			(* If we lose Side A Clamp PS In the AutoCycle between AC_Clamp and AC_Unclamp we Fault *)
			IF nActiveFaults[2].31=0 AND (nAutoCycleStep > AC_Clamp) AND ( nAutoCycleStep < AC_Unclamp) AND
				NOT bPS617
			THEN
				nActiveFaults[2].31:=1;
				IF (nFaultArrayIndex<=5) THEN
					arrFaultMessage[nFaultArrayIndex]:='F256 - Clamp Pressure Lost - Side A';
					arrFaultWarningCurrent[nCurrent]:='F256 - Clamp Pressure Lost - Side A';
					nFaultArrayIndex:=nFaultArrayIndex+1;
					nCurrent:=nCurrent+1;
				END_IF
			END_IF

		END_IF (*	Side A Faults *)

	(* 	SIDE B FAULTS
		The text of the fault comes from the function block "Side_B_Fixture" and we assign the hundreds series # to it below.
		Example: Side A Fixture has F2 is concated to the front of the text so that they are 200 series faults
				Side B fixture has F3 concated to make them 300 series faults..  
		You must go to the function block to see the rest of the number and the description text of the fault. 
		Generally this will be at the bottom of the function block. 	*)
		IF bSideBEnabled THEN
			(* Tailstock Side A *)
			IF nActiveFaults[3].0=0 AND Side_B_Fixture.bError THEN
				nActiveFaults[3].0:=1;
				IF (nFaultArrayIndex<=5) THEN
					arrFaultMessage[nFaultArrayIndex]:=CONCAT('F3',Side_B_Fixture.sErrorText);
						arrFaultMessage[nFaultArrayIndex]:=CONCAT(arrFaultMessage[nFaultArrayIndex],' Side B');
					arrFaultWarningCurrent[nCurrent]:=CONCAT('F3',Side_B_Fixture.sErrorText);
						arrFaultWarningCurrent[nCurrent]:=CONCAT(arrFaultWarningCurrent[nCurrent],' Side B');
					nCurrent:=nCurrent+1;
					nFaultArrayIndex:=nFaultArrayIndex+1;
					nCurrent:=nCurrent+1;
				END_IF
			END_IF

			IF nActiveFaults[3].1=0 AND bBCoolantSolenoid
				AND bLowFlow1B AND NOT(fCoolantFlowMin<0.5)
				AND fbFlowAverageTimer1BLOW.Q AND fbCoolantOnDelayTON.Q
			THEN
				nActiveFaults[3].1:=1;
				IF (nFaultArrayIndex<=5) THEN
					arrFaultMessage[nFaultArrayIndex]:='F330 - Coolant Flow Below Min #1B';
					arrFaultWarningCurrent[nCurrent]:='F330 - Coolant Flow Below Min #1B';
					nFaultArrayIndex:=nFaultArrayIndex+1;
					nCurrent:=nCurrent+1;
				END_IF
			END_IF
			IF nActiveFaults[3].2=0 AND bBCoolantSolenoid
				AND bHighFlow1B AND NOT(fCoolantFlowMax=60)
				AND fbFlowAverageTimer1BHIGH.Q AND fbCoolantOnDelayTON.Q
			THEN
				nActiveFaults[3].2:=1;
				IF (nFaultArrayIndex<=5) THEN
					arrFaultMessage[nFaultArrayIndex]:='F331 - Coolant Flow Exceeded Max #1B';
					arrFaultWarningCurrent[nCurrent]:='F331 - Coolant Flow Exceeded Max #1B';
					nFaultArrayIndex:=nFaultArrayIndex+1;
					nCurrent:=nCurrent+1;
				END_IF
			END_IF

			IF nActiveFaults[3].3=0 AND bBCoolantSolenoid
				AND bLowFlow2B AND NOT(fCoolantFlowMin<0.5)
				AND fbFlowAverageTimer2BLOW.Q AND fbCoolantOnDelayTON.Q
			THEN
				nActiveFaults[3].3:=1;
				IF (nFaultArrayIndex<=5) THEN
					arrFaultMessage[nFaultArrayIndex]:='F332 - Coolant Flow Below Min #2B';
					arrFaultWarningCurrent[nCurrent]:='F332 - Coolant Flow Below Min #2B';
					nFaultArrayIndex:=nFaultArrayIndex+1;
					nCurrent:=nCurrent+1;
				END_IF
			END_IF
			IF nActiveFaults[3].4=0 AND bBCoolantSolenoid
				AND bHighFlow2B AND NOT(fCoolantFlowMax=60)
				AND fbFlowAverageTimer2BHIGH.Q AND fbCoolantOnDelayTON.Q
			THEN
				nActiveFaults[3].4:=1;
				IF (nFaultArrayIndex<=5) THEN
					arrFaultMessage[nFaultArrayIndex]:='F333 - Coolant Flow Exceeded Max #2B';
					arrFaultWarningCurrent[nCurrent]:='F333 - Coolant Flow Exceeded Max #2B';
					nFaultArrayIndex:=nFaultArrayIndex+1;
					nCurrent:=nCurrent+1;
				END_IF
			END_IF

			IF nActiveFaults[3].5=0 AND bBCoolantSolenoid
				AND bLowFlow3B AND NOT(fCoolantFlowMin<0.5)
				AND fbFlowAverageTimer3BLOW.Q AND fbCoolantOnDelayTON.Q
			THEN
				nActiveFaults[3].5:=1;
				IF (nFaultArrayIndex<=5) THEN
					arrFaultMessage[nFaultArrayIndex]:='F334 - Coolant Flow Below Min #3B';
					arrFaultWarningCurrent[nCurrent]:='F334 - Coolant Flow Below Min #3B';
					nFaultArrayIndex:=nFaultArrayIndex+1;
					nCurrent:=nCurrent+1;
				END_IF
			END_IF
			IF nActiveFaults[3].6=0 AND bBCoolantSolenoid
				AND bHighFlow3B AND NOT(fCoolantFlowMax=60)
				AND fbFlowAverageTimer3BHIGH.Q AND fbCoolantOnDelayTON.Q
			THEN
				nActiveFaults[3].6:=1;
				IF (nFaultArrayIndex<=5) THEN
					arrFaultMessage[nFaultArrayIndex]:='F335 - Coolant Flow Exceeded Max #3B';
					arrFaultWarningCurrent[nCurrent]:='F335 - Coolant Flow Exceeded Max #3B';
					nFaultArrayIndex:=nFaultArrayIndex+1;
					nCurrent:=nCurrent+1;
				END_IF
			END_IF

			IF nActiveFaults[3].7=0 AND NOT(nServoThrustMax=0) AND fbServoBThrustMaxDelayTON.Q
				AND bInCycle AND NOT(stZBAxis.Status.InPositionArea) AND (stZBAxis.NcToPlc.AxisState=3) THEN
				nActiveFaults[3].7:=1;
				IF (nFaultArrayIndex<=5) THEN
					arrFaultMessage[nFaultArrayIndex]:='F336 - Servo ZB Thrust Exceeded Max';
					arrFaultWarningCurrent[nCurrent]:='F336 - Servo  ZBThrust Exceeded Max';
					nFaultArrayIndex:=nFaultArrayIndex+1;
					nCurrent:=nCurrent+1;
				END_IF
			END_IF

			IF nActiveFaults[3].8=0 AND stZBAxis.Status.Error  THEN
				nActiveFaults[3].8:=1;
				IF (nFaultArrayIndex<=5) THEN
					IF nZBAxisDiagNumber=64720 THEN
						arrFaultMessage[nFaultArrayIndex]:='F337a - ZB Negative Overtravel - (-) Motion Disabled';
						arrFaultWarningCurrent[nCurrent]:='F337a - ZB Negative Overtravel - (-) Motion Disabled';
					ELSIF nZBAxisDiagNumber=64721 THEN
						arrFaultMessage[nFaultArrayIndex]:='F337b - ZB Positive Overtravel - (+) Motion Disabled';
						arrFaultWarningCurrent[nCurrent]:='F337b - ZB Positive Overtravel - (+) Motion Disabled';
					ELSE
						arrFaultMessage[nFaultArrayIndex]:=CONCAT('F337 - Servo ZB Axis Fault# ',
							UDINT_TO_STRING(stZBAxis.Status.ErrorID));
						arrFaultWarningCurrent[nCurrent]:=CONCAT('F337 - Servo ZB Axis Fault# ',
							UDINT_TO_STRING(stZBAxis.Status.ErrorID));
					END_IF
					nFaultArrayIndex:=nFaultArrayIndex+1;
					nCurrent:=nCurrent+1;
				END_IF
			END_IF

			IF nActiveFaults[3].9=0 AND stWBAxis.Status.Error  THEN
				nActiveFaults[3].9:=1;
				IF (nFaultArrayIndex<=5) THEN
					IF nWBAxisDiagNumber=64720 THEN
						arrFaultMessage[nFaultArrayIndex]:='F338a - WB Negative Overtravel - (-) Motion Disabled';
						arrFaultWarningCurrent[nCurrent]:='F338a - WB Negative Overtravel - (-) Motion Disabled';
					ELSIF nWBAxisDiagNumber=64721 THEN
						arrFaultMessage[nFaultArrayIndex]:='F338b - WB Positive Overtravel - (+) Motion Disabled';
						arrFaultWarningCurrent[nCurrent]:='F338b - WB Positive Overtravel - (+) Motion Disabled';
					ELSE
						arrFaultMessage[nFaultArrayIndex]:=CONCAT('F338 - Servo WB Axis Fault# ',
							UDINT_TO_STRING(stWBAxis.Status.ErrorID));
						arrFaultWarningCurrent[nCurrent]:=CONCAT('F338 - Servo WB Axis Fault# ',
							UDINT_TO_STRING(stWBAxis.Status.ErrorID));
					END_IF
					nFaultArrayIndex:=nFaultArrayIndex+1;
					nCurrent:=nCurrent+1;
				END_IF
			END_IF

			IF nActiveFaults[3].10=0 AND fbHomeWB.Error  THEN
				nActiveFaults[3].10:=1;
				IF (nFaultArrayIndex<=5) THEN
					arrFaultMessage[nFaultArrayIndex]:='F339 - Tailstock WB Homing Error';
					arrFaultWarningCurrent[nCurrent]:='F339 - Tailstock WB Homing Error';;
					nFaultArrayIndex:=nFaultArrayIndex+1;
					nCurrent:=nCurrent+1;
				END_IF
			END_IF

			IF nActiveFaults[3].11=0 AND nSpindleLoad1BDisplay>nSpindleLoadMax AND NOT(nSpindleLoadMax=0)
				AND bVFD_BRun AND bVFD_B1UpToSpeed AND fbBLoadFaultDelay.Q THEN
				 nActiveFaults[3].11:=1;
				IF (nFaultArrayIndex<=5) THEN
					arrFaultMessage[nFaultArrayIndex]:='F340 - Spindle #1B Max Load Exceeded';
					arrFaultWarningCurrent[nCurrent]:='F340 - Spindle #1B Max Load Exceeded';
					nFaultArrayIndex:=nFaultArrayIndex+1;
					nCurrent:=nCurrent+1;
				END_IF
			END_IF

			IF nActiveFaults[3].12=0 AND nSpindleLoad2BDisplay>nSpindleLoadMax AND NOT(nSpindleLoadMax=0)
				AND bVFD_BRun AND bVFD_B2UpToSpeed AND fbBLoadFaultDelay.Q THEN
				 nActiveFaults[3].12:=1;
				IF (nFaultArrayIndex<=5) THEN
					arrFaultMessage[nFaultArrayIndex]:='F341 - Spindle #2B Max Load Exceeded';
					arrFaultWarningCurrent[nCurrent]:='F341 - Spindle #2B Max Load Exceeded';
					nFaultArrayIndex:=nFaultArrayIndex+1;
					nCurrent:=nCurrent+1;
				END_IF
			END_IF

			IF nActiveFaults[3].13=0 AND nSpindleLoad3BDisplay>nSpindleLoadMax AND NOT(nSpindleLoadMax=0)
				AND bVFD_BRun AND bVFD_B3UpToSpeed AND fbBLoadFaultDelay.Q THEN
				 nActiveFaults[3].13:=1;
				IF (nFaultArrayIndex<=5) THEN
					arrFaultMessage[nFaultArrayIndex]:='F342 - Spindle #3B Max Load Exceeded';
					arrFaultWarningCurrent[nCurrent]:='F342 - Spindle #3B Max Load Exceeded';
					nFaultArrayIndex:=nFaultArrayIndex+1;
					nCurrent:=nCurrent+1;
				END_IF
			END_IF

	(* Spares *)

			IF nActiveFaults[3].18=0 AND fbVFD_B1.bError THEN
			(*	Encompasses ALL VFD related Errors *)
			(* uptospeed, drivenotready, drivefaulted, drivewarning, drivecomm *)
				nActiveFaults[3].18:=1;
				IF (nFaultArrayIndex<=5) THEN
					IF fbVFD_B1.nErrorID=Er_DriveComm THEN
						arrFaultMessage[nFaultArrayIndex]:='F343a - Spindle #1B VFD Communcation Failed';
						arrFaultWarningCurrent[nCurrent]:='F343a - Spindle #1B VFD Communcation Failed';
						nFaultArrayIndex:=nFaultArrayIndex+1;
						nCurrent:=nCurrent+1;
					ELSIF fbVFD_B1.nErrorID=Er_DriveFaulted THEN
						arrFaultMessage[nFaultArrayIndex]:='F343b - Spindle #1B VFD Fault';
						arrFaultWarningCurrent[nCurrent]:='F343b - Spindle #1B VFD Fault';
						nFaultArrayIndex:=nFaultArrayIndex+1;
						nCurrent:=nCurrent+1;
					ELSIF fbVFD_B1.nErrorID=Er_DriveWarning THEN
						arrFaultMessage[nFaultArrayIndex]:='F343c - Spindle #1B VFD Warning';
						arrFaultWarningCurrent[nCurrent]:='F343c - Spindle #1B VFD Warning';
						nFaultArrayIndex:=nFaultArrayIndex+1;
						nCurrent:=nCurrent+1;
					ELSIF fbVFD_B1.nErrorID=Er_DriveNotReady THEN
						arrFaultMessage[nFaultArrayIndex]:='F343d - Spindle #1B VFD Not Ready';
						arrFaultWarningCurrent[nCurrent]:='F343d - Spindle #1B VFD Not Ready';
						nFaultArrayIndex:=nFaultArrayIndex+1;
						nCurrent:=nCurrent+1;
					ELSIF fbVFD_B1.nErrorID=Er_InvalidRPM THEN
						arrFaultMessage[nFaultArrayIndex]:='F343e - Spindle #1B VFD Invalid RPM Requested';
						arrFaultWarningCurrent[nCurrent]:='F343e - Spindle #1B VFD Invalid RPM Requested';
						nFaultArrayIndex:=nFaultArrayIndex+1;
						nCurrent:=nCurrent+1;
					ELSIF fbVFD_B1.nErrorID=Er_InvalidRatio THEN
						arrFaultMessage[nFaultArrayIndex]:='F343f - Spindle #1B VFD Invalid Motor to Spindle Ratio Requested';
						arrFaultWarningCurrent[nCurrent]:='F343f - Spindle #1B VFD Invalid Motor to Spindle Ratio Requested';
						nFaultArrayIndex:=nFaultArrayIndex+1;
						nCurrent:=nCurrent+1;
					ELSIF fbVFD_B1.nErrorID=Er_InvalidOverride THEN
						arrFaultMessage[nFaultArrayIndex]:='F343g - Spindle #1B VFD Invalid Override Requested';
						arrFaultWarningCurrent[nCurrent]:='F343g - Spindle #1B VFD Invalid Override Requested';
						nFaultArrayIndex:=nFaultArrayIndex+1;
						nCurrent:=nCurrent+1;
					ELSIF fbVFD_B1.nErrorID=Er_UpToSpeedTimeout THEN
						arrFaultMessage[nFaultArrayIndex]:='F343h - Spindle #1B VFD Not Up To Speed';
						arrFaultWarningCurrent[nCurrent]:='F343h - Spindle #1B VFD Not Up To Speed';
						nFaultArrayIndex:=nFaultArrayIndex+1;
						nCurrent:=nCurrent+1;
					ELSE
						arrFaultMessage[nFaultArrayIndex]:=CONCAT('F343 - Spindle #1B VFD Error : ',
												UDINT_TO_STRING(fbVFD_B1.stVFDInfo.nActiveFault));
						arrFaultWarningCurrent[nCurrent]:=CONCAT('F343 - Spindle #1B VFD Error : ',
												UDINT_TO_STRING(fbVFD_B1.stVFDInfo.nActiveFault));
						nFaultArrayIndex:=nFaultArrayIndex+1;
						nCurrent:=nCurrent+1;
					END_IF
				END_IF
			END_IF

			IF nActiveFaults[3].19=0 AND fbVFD_B2.bError THEN
			(*	Encompasses ALL VFD related Errors *)
			(* uptospeed, drivenotready, drivefaulted, drivewarning, drivecomm *)
				nActiveFaults[3].19:=1;
				IF (nFaultArrayIndex<=5) THEN
					IF fbVFD_B2.nErrorID=Er_DriveComm THEN
						arrFaultMessage[nFaultArrayIndex]:='F344a - Spindle #2B VFD Communcation Failed';
						arrFaultWarningCurrent[nCurrent]:='F344a - Spindle #2B VFD Communcation Failed';
						nFaultArrayIndex:=nFaultArrayIndex+1;
						nCurrent:=nCurrent+1;
					ELSIF fbVFD_B2.nErrorID=Er_DriveFaulted THEN
						arrFaultMessage[nFaultArrayIndex]:='F344b - Spindle #2B VFD Fault';
						arrFaultWarningCurrent[nCurrent]:='F344b - Spindle #2B VFD Fault';
						nFaultArrayIndex:=nFaultArrayIndex+1;
						nCurrent:=nCurrent+1;
					ELSIF fbVFD_B2.nErrorID=Er_DriveWarning THEN
						arrFaultMessage[nFaultArrayIndex]:='F344c - Spindle #2B VFD Warning';
						arrFaultWarningCurrent[nCurrent]:='F344c - Spindle #2B VFD Warning';
						nFaultArrayIndex:=nFaultArrayIndex+1;
						nCurrent:=nCurrent+1;
					ELSIF fbVFD_B2.nErrorID=Er_DriveNotReady THEN
						arrFaultMessage[nFaultArrayIndex]:='F344d - Spindle #2B VFD Not Ready';
						arrFaultWarningCurrent[nCurrent]:='F344d - Spindle #2B VFD Not Ready';
						nFaultArrayIndex:=nFaultArrayIndex+1;
						nCurrent:=nCurrent+1;
					ELSIF fbVFD_B2.nErrorID=Er_InvalidRPM THEN
						arrFaultMessage[nFaultArrayIndex]:='F344e - Spindle #2B VFD Invalid RPM Requested';
						arrFaultWarningCurrent[nCurrent]:='F344e - Spindle #2B VFD Invalid RPM Requested';
						nFaultArrayIndex:=nFaultArrayIndex+1;
						nCurrent:=nCurrent+1;
					ELSIF fbVFD_B2.nErrorID=Er_InvalidRatio THEN
						arrFaultMessage[nFaultArrayIndex]:='F344f - Spindle #2B VFD Invalid Motor to Spindle Ratio Requested';
						arrFaultWarningCurrent[nCurrent]:='F344f - Spindle #2B VFD Invalid Motor to Spindle Ratio Requested';
						nFaultArrayIndex:=nFaultArrayIndex+1;
						nCurrent:=nCurrent+1;
					ELSIF fbVFD_B2.nErrorID=Er_InvalidOverride THEN
						arrFaultMessage[nFaultArrayIndex]:='F344g - Spindle #2B VFD Invalid Override Requested';
						arrFaultWarningCurrent[nCurrent]:='F344g - Spindle #2B VFD Invalid Override Requested';
						nFaultArrayIndex:=nFaultArrayIndex+1;
						nCurrent:=nCurrent+1;
					ELSIF fbVFD_B2.nErrorID=Er_UpToSpeedTimeout THEN
						arrFaultMessage[nFaultArrayIndex]:='F344h - Spindle #2B VFD Not Up To Speed';
						arrFaultWarningCurrent[nCurrent]:='F344h - Spindle #2B VFD Not Up To Speed';
						nFaultArrayIndex:=nFaultArrayIndex+1;
						nCurrent:=nCurrent+1;
					ELSE
						arrFaultMessage[nFaultArrayIndex]:=CONCAT('F344 - Spindle #2B VFD Error : ',
												UDINT_TO_STRING(fbVFD_B2.stVFDInfo.nActiveFault));
						arrFaultWarningCurrent[nCurrent]:=CONCAT('F344 - Spindle #2B VFD Error : ',
												UDINT_TO_STRING(fbVFD_B2.stVFDInfo.nActiveFault));
						nFaultArrayIndex:=nFaultArrayIndex+1;
						nCurrent:=nCurrent+1;
					END_IF
				END_IF
			END_IF

			IF nActiveFaults[3].20=0 AND fbVFD_B3.bError THEN
			(*	Encompasses ALL VFD related Errors *)
			(* uptospeed, drivenotready, drivefaulted, drivewarning, drivecomm *)
				nActiveFaults[3].20:=1;
				IF (nFaultArrayIndex<=5) THEN
					IF fbVFD_B3.nErrorID=Er_DriveComm THEN
						arrFaultMessage[nFaultArrayIndex]:='F345a - Spindle #3B VFD Communcation Failed';
						arrFaultWarningCurrent[nCurrent]:='F345a - Spindle #3B VFD Communcation Failed';
						nFaultArrayIndex:=nFaultArrayIndex+1;
						nCurrent:=nCurrent+1;
					ELSIF fbVFD_B3.nErrorID=Er_DriveFaulted THEN
						arrFaultMessage[nFaultArrayIndex]:='F345b - Spindle #3B VFD Fault';
						arrFaultWarningCurrent[nCurrent]:='F345b - Spindle #3B VFD Fault';
						nFaultArrayIndex:=nFaultArrayIndex+1;
						nCurrent:=nCurrent+1;
					ELSIF fbVFD_B3.nErrorID=Er_DriveWarning THEN
						arrFaultMessage[nFaultArrayIndex]:='F345c - Spindle #3B VFD Warning';
						arrFaultWarningCurrent[nCurrent]:='F345c - Spindle #3B VFD Warning';
						nFaultArrayIndex:=nFaultArrayIndex+1;
						nCurrent:=nCurrent+1;
					ELSIF fbVFD_B3.nErrorID=Er_DriveNotReady THEN
						arrFaultMessage[nFaultArrayIndex]:='F345d - Spindle #3B VFD Not Ready';
						arrFaultWarningCurrent[nCurrent]:='F345d - Spindle #3B VFD Not Ready';
						nFaultArrayIndex:=nFaultArrayIndex+1;
						nCurrent:=nCurrent+1;
					ELSIF fbVFD_B3.nErrorID=Er_InvalidRPM THEN
						arrFaultMessage[nFaultArrayIndex]:='F345e - Spindle #3B VFD Invalid RPM Requested';
						arrFaultWarningCurrent[nCurrent]:='F345e - Spindle #3B VFD Invalid RPM Requested';
						nFaultArrayIndex:=nFaultArrayIndex+1;
						nCurrent:=nCurrent+1;
					ELSIF fbVFD_B3.nErrorID=Er_InvalidRatio THEN
						arrFaultMessage[nFaultArrayIndex]:='F345f - Spindle #3B VFD Invalid Motor to Spindle Ratio Requested';
						arrFaultWarningCurrent[nCurrent]:='F345f - Spindle #3B VFD Invalid Motor to Spindle Ratio Requested';
						nFaultArrayIndex:=nFaultArrayIndex+1;
						nCurrent:=nCurrent+1;
					ELSIF fbVFD_B3.nErrorID=Er_InvalidOverride THEN
						arrFaultMessage[nFaultArrayIndex]:='F345g - Spindle #3B VFD Invalid Override Requested';
						arrFaultWarningCurrent[nCurrent]:='F345g - Spindle #3B VFD Invalid Override Requested';
						nFaultArrayIndex:=nFaultArrayIndex+1;
						nCurrent:=nCurrent+1;
					ELSIF fbVFD_B3.nErrorID=Er_UpToSpeedTimeout THEN
						arrFaultMessage[nFaultArrayIndex]:='F345h - Spindle #3B VFD Not Up To Speed';
						arrFaultWarningCurrent[nCurrent]:='F345h - Spindle #3B VFD Not Up To Speed';
						nFaultArrayIndex:=nFaultArrayIndex+1;
						nCurrent:=nCurrent+1;
					ELSE
						arrFaultMessage[nFaultArrayIndex]:=CONCAT('F345 - Spindle #3B VFD Error : ',
												UDINT_TO_STRING(fbVFD_B3.stVFDInfo.nActiveFault));
						arrFaultWarningCurrent[nCurrent]:=CONCAT('F345 - Spindle #3B VFD Error : ',
												UDINT_TO_STRING(fbVFD_B3.stVFDInfo.nActiveFault));
						nFaultArrayIndex:=nFaultArrayIndex+1;
						nCurrent:=nCurrent+1;
					END_IF
				END_IF
			END_IF

			(* Coolant Pressure Fault for Auto Mode *)
			IF nActiveFaults[3].21=0 AND fbLowPressureFaultBDelay.Q
				AND bMachineMode
			THEN
				nActiveFaults[3].21:=1;
				IF (nFaultArrayIndex<=5) THEN
					arrFaultMessage[nFaultArrayIndex]:='F346 - Coolant Pressure Low - Side B';
					arrFaultWarningCurrent[nCurrent]:='F346 - Coolant Pressure Low - Side B';
					nFaultArrayIndex:=nFaultArrayIndex+1;
					nCurrent:=nCurrent+1;
				END_IF
			END_IF

			IF nActiveFaults[3].22=0 AND fbSpeedVariationTimer1BHIGH.Q
				AND bVFD_BRun  AND bVFD_B1UpToSpeed AND (bInCycle OR bSetupB)
				AND fbBSpeedDelayTimer.Q THEN
				nActiveFaults[3].22:=1;
				IF (nFaultArrayIndex<=5) THEN
					arrFaultMessage[nFaultArrayIndex]:='F347 - Spindle Speed Not Correct #1B (HIGH)';
					arrFaultWarningCurrent[nCurrent]:='F333 - Spindle Speed Not Correct #1B (HIGH)';
					nFaultArrayIndex:=nFaultArrayIndex+1;
					nCurrent:=nCurrent+1;
				END_IF
			END_IF
			IF nActiveFaults[3].23=0 AND fbSpeedVariationTimer1BLOW.Q
				AND bVFD_BRun AND bVFD_B1UpToSpeed AND (bInCycle OR bSetupB)
				AND fbBSpeedDelayTimer.Q THEN
				nActiveFaults[3].23:=1;
				IF (nFaultArrayIndex<=5) THEN
					arrFaultMessage[nFaultArrayIndex]:='F348 - Spindle Speed Not Correct #1B (LOW)';
					arrFaultWarningCurrent[nCurrent]:='F348 - Spindle Speed Not Correct #1B (LOW)';
					nFaultArrayIndex:=nFaultArrayIndex+1;
					nCurrent:=nCurrent+1;
				END_IF
			END_IF

			IF nActiveFaults[3].24=0 AND fbSpeedVariationTimer2BHIGH.Q
				AND bVFD_BRun  AND bVFD_B2UpToSpeed AND (bInCycle OR bSetupB)
				AND fbBSpeedDelayTimer.Q THEN
				nActiveFaults[3].24:=1;
				IF (nFaultArrayIndex<=5) THEN
					arrFaultMessage[nFaultArrayIndex]:='F349 - Spindle Speed Not Correct #2B (HIGH)';
					arrFaultWarningCurrent[nCurrent]:='F349 - Spindle Speed Not Correct #2B (HIGH)';
					nFaultArrayIndex:=nFaultArrayIndex+1;
					nCurrent:=nCurrent+1;
				END_IF
			END_IF

			IF nActiveFaults[3].25=0 AND fbSpeedVariationTimer2BLOW.Q
				AND bVFD_BRun AND bVFD_B2UpToSpeed AND (bInCycle OR bSetupB)
				AND fbBSpeedDelayTimer.Q THEN
				nActiveFaults[3].25:=1;
				IF (nFaultArrayIndex<=5) THEN
					arrFaultMessage[nFaultArrayIndex]:='F350 - Spindle Speed Not Correct #2B (LOW)';
					arrFaultWarningCurrent[nCurrent]:='F350 - Spindle Speed Not Correct #2B (LOW)';
					nFaultArrayIndex:=nFaultArrayIndex+1;
					nCurrent:=nCurrent+1;
				END_IF
			END_IF

			IF nActiveFaults[3].26=0 AND fbSpeedVariationTimer3BHIGH.Q
				AND bVFD_BRun  AND bVFD_B3UpToSpeed AND (bInCycle OR bSetupB)
				AND fbBSpeedDelayTimer.Q THEN
				nActiveFaults[3].26:=1;
				IF (nFaultArrayIndex<=5) THEN
					arrFaultMessage[nFaultArrayIndex]:='F351 - Spindle Speed Not Correct #3B (HIGH)';
					arrFaultWarningCurrent[nCurrent]:='F351 - Spindle Speed Not Correct #3B (HIGH)';
					nFaultArrayIndex:=nFaultArrayIndex+1;
					nCurrent:=nCurrent+1;
				END_IF
			END_IF

			IF nActiveFaults[3].27=0 AND fbSpeedVariationTimer3BLOW.Q
				AND bVFD_BRun AND bVFD_B3UpToSpeed AND (bInCycle OR bSetupB)
				AND fbBSpeedDelayTimer.Q THEN
				nActiveFaults[3].27:=1;
				IF (nFaultArrayIndex<=5) THEN
					arrFaultMessage[nFaultArrayIndex]:='F352 - Spindle Speed Not Correct #3B (LOW)';
					arrFaultWarningCurrent[nCurrent]:='F352 - Spindle Speed Not Correct #3B (LOW)';
					nFaultArrayIndex:=nFaultArrayIndex+1;
					nCurrent:=nCurrent+1;
				END_IF
			END_IF

			IF nActiveFaults[3].28=0 AND nModeError=Er_SideBColletSolError THEN
				nModeError:=Er_NoModeError;
				nActiveFaults[3].28:=1;
				IF (nFaultArrayIndex<=5) THEN
					arrFaultMessage[nFaultArrayIndex]:='F353 - Both B Clamp and UnClamp Solenoids On At Same Time';
					arrFaultWarningCurrent[nCurrent]:='F353 - Both B Clamp and UnClamp Solenoids On At Same Time';
					nFaultArrayIndex:=nFaultArrayIndex+1;
					nCurrent:=nCurrent+1;
				END_IF
			END_IF

			IF nActiveFaults[3].29=0 AND nModeError=Er_SideBEjectorsSolError THEN
				nModeError:=Er_NoModeError;
				nActiveFaults[3].29:=1;
				IF (nFaultArrayIndex<=5) THEN
					arrFaultMessage[nFaultArrayIndex]:='F354 - Both B Ejector Advance  and Retract Solenoids On At Same Time';
					arrFaultWarningCurrent[nCurrent]:='F354 - Both B Ejector Advance  and Retract Solenoids On At Same Time';
					nFaultArrayIndex:=nFaultArrayIndex+1;
					nCurrent:=nCurrent+1;
				END_IF
			END_IF

			IF nActiveFaults[3].30=0 AND bRack7Comm THEN
				nActiveFaults[3].30:=1;
				IF (nFaultArrayIndex<=5) THEN
					arrFaultMessage[nFaultArrayIndex]:='F355 - Com. Lost to Side B Tailstock Input Module';
					arrFaultWarningCurrent[nCurrent]:='F355 - Com. Lost to Side B Tailstock Input Module';
					nFaultArrayIndex:=nFaultArrayIndex+1;
					nCurrent:=nCurrent+1;
				END_IF
			END_IF

			(* If we lose Side B Clamp PS In the AutoCycle between AC_Clamp and AC_Unclamp we Fault *)
			IF nActiveFaults[3].31=0 AND (nAutoCycleStep > AC_Clamp) AND (nAutoCycleStep < AC_Unclamp) AND
				NOT bPS727
			THEN
				nActiveFaults[3].31:=1;
				IF (nFaultArrayIndex<=5) THEN
					arrFaultMessage[nFaultArrayIndex]:='F356 - Clamp Pressure Lost - Side B';
					arrFaultWarningCurrent[nCurrent]:='F356 - Clamp Pressure Lost - Side B';
					nFaultArrayIndex:=nFaultArrayIndex+1;
					nCurrent:=nCurrent+1;
				END_IF
			END_IF

		END_IF (*	Side B Faults *)

	(* Faults that do not Stop a Drilling Cycle *)

		IF nActiveFaults[4].0=0 AND bFilter1Dirty AND nDirtyCount1=5 THEN
			nActiveFaults[4].0:=1;
			IF (nFaultArrayIndex<=5) THEN
				arrFaultMessage[nFaultArrayIndex]:='F400 - Filter #1 Clogged (MUST CHANGE)';
				arrFaultWarningCurrent[nCurrent]:='F400 - Filter #1 Clogged (MUST CHANGE)';
				nFaultArrayIndex:=nFaultArrayIndex+1;
				nCurrent:=nCurrent+1;
			END_IF
		END_IF

		IF nActiveFaults[4].1=0 AND bFilter2Dirty AND nDirtyCount2=5 THEN
			nActiveFaults[4].1:=1;
			IF (nFaultArrayIndex<=5) THEN
				arrFaultMessage[nFaultArrayIndex]:='F401 - Filter #2 Clogged (MUST CHANGE)';
				arrFaultWarningCurrent[nCurrent]:='F401 - Filter #2 Clogged (MUST CHANGE)';
				nFaultArrayIndex:=nFaultArrayIndex+1;
				nCurrent:=nCurrent+1;
			END_IF
		END_IF

		IF nActiveFaults[4].2=0 AND bFilter3Dirty AND nDirtyCount3=5 THEN
			nActiveFaults[4].2:=1;
			IF (nFaultArrayIndex<=5) THEN
				arrFaultMessage[nFaultArrayIndex]:='F402 - Filter #3 Clogged (MUST CHANGE)';
				arrFaultWarningCurrent[nCurrent]:='F402 - Filter #3 Clogged (MUST CHANGE)';
				nFaultArrayIndex:=nFaultArrayIndex+1;
				nCurrent:=nCurrent+1;
			END_IF
		END_IF

		IF nActiveFaults[4].3=0 AND bFilter4Dirty AND nDirtyCount4=5 THEN
			nActiveFaults[4].3:=1;
			IF (nFaultArrayIndex<=5) THEN
				arrFaultMessage[nFaultArrayIndex]:='F403 - Filter #4 Clogged (MUST CHANGE)';
				arrFaultWarningCurrent[nCurrent]:='F403 - Filter #4 Clogged (MUST CHANGE)';
				nFaultArrayIndex:=nFaultArrayIndex+1;
				nCurrent:=nCurrent+1;
			END_IF
		END_IF

		IF nActiveFaults[4].4=0 AND NOT(bLubeLevel) AND (nLubeLevelLowCount>=3) THEN
			nActiveFaults[4].4:=1;
			IF (nFaultArrayIndex<=5) THEN
				arrFaultMessage[nFaultArrayIndex]:='F404 - Lube Level Low (MUST FILL)';
				arrFaultWarningCurrent[nCurrent]:='F404 - Lube Level Low (MUST FILL)';
				nFaultArrayIndex:=nFaultArrayIndex+1;
				nCurrent:=nCurrent+1;
			END_IF
		END_IF

		(* Fault if Side A Collet Clamped and X selected on MPG *)
		IF nActiveFaults[4].5=0 AND ( ( (bPS617 OR bATailstockColletClamp) AND bXAAxisSelected) OR
			( (bPS727 OR bBTailstockColletClamp) AND bXBAxisSelected) ) THEN
			nActiveFaults[4].5:=1;
			IF (nFaultArrayIndex<=5) THEN
				IF bXAAxisSelected THEN
					arrFaultMessage[nFaultArrayIndex]:='F405A - MPG XA Selected While Clamped';
					arrFaultWarningCurrent[nCurrent]:='F405A - MPG XA Selected While Clamped';
				ELSE
					arrFaultMessage[nFaultArrayIndex]:='F405B - MPG XB Selected While Clamped';
					arrFaultWarningCurrent[nCurrent]:='F405B - MPG XB Selected While Clamped';
				END_IF
				nFaultArrayIndex:=nFaultArrayIndex+1;
				nCurrent:=nCurrent+1;
			END_IF
		END_IF

		(* Fault if Side A Collet Clamped and ZA or WA selected on MPG *)
		IF nActiveFaults[4].6=0 AND (bPS617 OR bATailstockColletClamp) AND (bZAAxisSelected OR bWAAxisSelected) THEN
			nActiveFaults[4].6:=1;
			IF (nFaultArrayIndex<=5) THEN
				arrFaultMessage[nFaultArrayIndex]:='F406 - MPG ZA or WA Selected While Clamped';
				arrFaultWarningCurrent[nCurrent]:='F406 - MPG ZA or WA Selected While Clamped';
				nFaultArrayIndex:=nFaultArrayIndex+1;
				nCurrent:=nCurrent+1;
			END_IF
		END_IF

		(* Fault if Side B Collet Clamped and ZB or WB selected on MPG *)
		IF nActiveFaults[4].7=0 AND (bPS727 OR bBTailstockColletClamp) AND (bZBAxisSelected OR bWBAxisSelected) THEN
			nActiveFaults[4].7:=1;
			IF (nFaultArrayIndex<=5) THEN
				arrFaultMessage[nFaultArrayIndex]:='F407 - MPG ZB or WB Selected While Clamped';
				arrFaultWarningCurrent[nCurrent]:='F407 - MPG ZB or WB Selected While Clamped';
				nFaultArrayIndex:=nFaultArrayIndex+1;
				nCurrent:=nCurrent+1;
			END_IF
		END_IF

	(* 	WARNINGS		*)

		IF nActiveWarnings[1].0=0 AND fbCoolantTempWarningTON.Q THEN
			nActiveWarnings[1].0:=1;
			IF (nWarningArrayIndex<=5) THEN
				arrFaultMessage[nWarningArrayIndex+5]:='W001 - Coolant Temperature Warning';
				arrFaultWarningCurrent[nCurrent]:='W001 - Coolant Temperature Warning';
				nWarningArrayIndex:=nWarningArrayIndex+1;
				nCurrent:=nCurrent+1;
			END_IF
		ELSIF NOT( bCoolantTempWarning) AND nActiveWarnings[1].0=1 THEN
			IF FIND(arrFaultMessage[6], 'W001')>0 THEN
				arrFaultMessage[6]:=arrFaultMessage[7];
				arrFaultMessage[7]:=arrFaultMessage[8];
				arrFaultMessage[8]:=arrFaultMessage[9];
				arrFaultMessage[9]:=arrFaultMessage[10];
				arrFaultMessage[10]:='';
				nActiveWarnings[1].0:=0;
				nWarningArrayIndex:=nWarningArrayIndex-1;
			ELSIF FIND(arrFaultMessage[7], 'W001')>0 THEN
				arrFaultMessage[7]:=arrFaultMessage[8];
				arrFaultMessage[8]:=arrFaultMessage[9];
				arrFaultMessage[9]:=arrFaultMessage[10];
				arrFaultMessage[10]:='';
				nActiveWarnings[1].0:=0;
				nWarningArrayIndex:=nWarningArrayIndex-1;
			ELSIF FIND(arrFaultMessage[8], 'W001')>0 THEN
				arrFaultMessage[8]:=arrFaultMessage[9];
				arrFaultMessage[9]:=arrFaultMessage[10];
				arrFaultMessage[10]:='';
				nActiveWarnings[1].0:=0;
				nWarningArrayIndex:=nWarningArrayIndex-1;
			ELSIF FIND(arrFaultMessage[9], 'W001')>0 THEN
				arrFaultMessage[9]:=arrFaultMessage[10];
				arrFaultMessage[10]:='';
				nActiveWarnings[1].0:=0;
				nWarningArrayIndex:=nWarningArrayIndex-1;
			ELSIF FIND(arrFaultMessage[10], 'W001')>0 THEN
				arrFaultMessage[10]:='';
				nActiveWarnings[1].0:=0;
				nWarningArrayIndex:=nWarningArrayIndex-1;
			ELSE
				nActiveWarnings[1].0:=0;
				nWarningArrayIndex:=nWarningArrayIndex-1;
			END_IF
		END_IF

		IF nActiveWarnings[1].1=0 AND NOT(bProx310)
			AND (bMachineMode OR bEnterAutoModePB) AND NOT(bInCycle) THEN
			nActiveWarnings[1].1:=1;
			IF (nWarningArrayIndex<=5) THEN
				arrFaultMessage[nWarningArrayIndex+5]:='W002 - Tool Change Door Open Side A';
				arrFaultWarningCurrent[nCurrent]:='W002 - Tool Change Door Open Side A';
				nWarningArrayIndex:=nWarningArrayIndex+1;
				nCurrent:=nCurrent+1;
			END_IF
		ELSIF bProx310 AND nActiveWarnings[1].1 THEN
			IF FIND(arrFaultMessage[6], 'W002')>0 THEN
				arrFaultMessage[6]:=arrFaultMessage[7];
				arrFaultMessage[7]:=arrFaultMessage[8];
				arrFaultMessage[8]:=arrFaultMessage[9];
				arrFaultMessage[9]:=arrFaultMessage[10];
				arrFaultMessage[10]:='';
				nActiveWarnings[1].1:=0;
				nWarningArrayIndex:=nWarningArrayIndex-1;
			ELSIF FIND(arrFaultMessage[7], 'W002')>0 THEN
				arrFaultMessage[7]:=arrFaultMessage[8];
				arrFaultMessage[8]:=arrFaultMessage[9];
				arrFaultMessage[9]:=arrFaultMessage[10];
				arrFaultMessage[10]:='';
				nActiveWarnings[1].1:=0;
				nWarningArrayIndex:=nWarningArrayIndex-1;
			ELSIF FIND(arrFaultMessage[8], 'W002')>0 THEN
				arrFaultMessage[8]:=arrFaultMessage[9];
				arrFaultMessage[9]:=arrFaultMessage[10];
				arrFaultMessage[10]:='';
				nActiveWarnings[1].1:=0;
				nWarningArrayIndex:=nWarningArrayIndex-1;
			ELSIF FIND(arrFaultMessage[9], 'W002')>0 THEN
				arrFaultMessage[9]:=arrFaultMessage[10];
				arrFaultMessage[10]:='';
				nActiveWarnings[1].1:=0;
				nWarningArrayIndex:=nWarningArrayIndex-1;
			ELSIF FIND(arrFaultMessage[10], 'W002')>0 THEN
				arrFaultMessage[10]:='';
				nActiveWarnings[1].1:=0;
				nWarningArrayIndex:=nWarningArrayIndex-1;
			ELSE
				nActiveWarnings[1].1:=0;
				nWarningArrayIndex:=nWarningArrayIndex-1;
			END_IF
		END_IF

		IF nActiveWarnings[1].2=0 AND NOT(bProx312)
			AND (bMachineMode OR bEnterAutoModePB) AND NOT(bInCycle) THEN
			nActiveWarnings[1].2:=1;
			IF (nWarningArrayIndex<=5) THEN
				arrFaultMessage[nWarningArrayIndex+5]:='W003 - Tailstock Door Open Side A';
				arrFaultWarningCurrent[nCurrent]:='W003 - Tailstock Door Open Side A';
				nWarningArrayIndex:=nWarningArrayIndex+1;
				nCurrent:=nCurrent+1;
			END_IF
		ELSIF bProx312 AND nActiveWarnings[1].2 THEN
			IF FIND(arrFaultMessage[6], 'W003')>0 THEN
				arrFaultMessage[6]:=arrFaultMessage[7];
				arrFaultMessage[7]:=arrFaultMessage[8];
				arrFaultMessage[8]:=arrFaultMessage[9];
				arrFaultMessage[9]:=arrFaultMessage[10];
				arrFaultMessage[10]:='';
				nActiveWarnings[1].2:=0;
				nWarningArrayIndex:=nWarningArrayIndex-1;
			ELSIF FIND(arrFaultMessage[7], 'W003')>0 THEN
				arrFaultMessage[7]:=arrFaultMessage[8];
				arrFaultMessage[8]:=arrFaultMessage[9];
				arrFaultMessage[9]:=arrFaultMessage[10];
				arrFaultMessage[10]:='';
				nActiveWarnings[1].2:=0;
				nWarningArrayIndex:=nWarningArrayIndex-1;
			ELSIF FIND(arrFaultMessage[8], 'W003')>0 THEN
				arrFaultMessage[8]:=arrFaultMessage[9];
				arrFaultMessage[9]:=arrFaultMessage[10];
				arrFaultMessage[10]:='';
				nActiveWarnings[1].2:=0;
				nWarningArrayIndex:=nWarningArrayIndex-1;
			ELSIF FIND(arrFaultMessage[9], 'W003')>0 THEN
				arrFaultMessage[9]:=arrFaultMessage[10];
				arrFaultMessage[10]:='';
				nActiveWarnings[1].2:=0;
				nWarningArrayIndex:=nWarningArrayIndex-1;
			ELSIF FIND(arrFaultMessage[10], 'W003')>0 THEN
				arrFaultMessage[10]:='';
				nActiveWarnings[1].2:=0;
				nWarningArrayIndex:=nWarningArrayIndex-1;
			ELSE
				nActiveWarnings[1].2:=0;
				nWarningArrayIndex:=nWarningArrayIndex-1;
			END_IF
		END_IF

		IF nActiveWarnings[1].3=0 AND NOT(bProx313)
			AND (bMachineMode OR bEnterAutoModePB) AND NOT(bInCycle) THEN
			nActiveWarnings[1].3:=1;
			IF (nWarningArrayIndex<=5) THEN
				arrFaultMessage[nWarningArrayIndex+5]:='W004 - Tailstock Door Open Side B';
				arrFaultWarningCurrent[nCurrent]:='W004 - Tailstock Door Open Side B';
				nWarningArrayIndex:=nWarningArrayIndex+1;
				nCurrent:=nCurrent+1;
			END_IF
		ELSIF bProx313 AND nActiveWarnings[1].3 THEN
			IF FIND(arrFaultMessage[6], 'W004')>0 THEN
				arrFaultMessage[6]:=arrFaultMessage[7];
				arrFaultMessage[7]:=arrFaultMessage[8];
				arrFaultMessage[8]:=arrFaultMessage[9];
				arrFaultMessage[9]:=arrFaultMessage[10];
				arrFaultMessage[10]:='';
				nActiveWarnings[1].3:=0;
				nWarningArrayIndex:=nWarningArrayIndex-1;
			ELSIF FIND(arrFaultMessage[7], 'W004')>0 THEN
				arrFaultMessage[7]:=arrFaultMessage[8];
				arrFaultMessage[8]:=arrFaultMessage[9];
				arrFaultMessage[9]:=arrFaultMessage[10];
				arrFaultMessage[10]:='';
				nActiveWarnings[1].3:=0;
				nWarningArrayIndex:=nWarningArrayIndex-1;
			ELSIF FIND(arrFaultMessage[8], 'W004')>0 THEN
				arrFaultMessage[8]:=arrFaultMessage[9];
				arrFaultMessage[9]:=arrFaultMessage[10];
				arrFaultMessage[10]:='';
				nActiveWarnings[1].3:=0;
				nWarningArrayIndex:=nWarningArrayIndex-1;
			ELSIF FIND(arrFaultMessage[9], 'W004')>0 THEN
				arrFaultMessage[9]:=arrFaultMessage[10];
				arrFaultMessage[10]:='';
				nActiveWarnings[1].3:=0;
				nWarningArrayIndex:=nWarningArrayIndex-1;
			ELSIF FIND(arrFaultMessage[10], 'W004')>0 THEN
				arrFaultMessage[10]:='';
				nActiveWarnings[1].3:=0;
				nWarningArrayIndex:=nWarningArrayIndex-1;
			ELSE
				nActiveWarnings[1].3:=0;
				nWarningArrayIndex:=nWarningArrayIndex-1;
			END_IF
		END_IF

		IF nActiveWarnings[1].4=0 AND fbFilter1Timer.Q AND nDirtyCount1<5 THEN
			nDirtyCount1:=nDirtyCount1+1;
			nActiveWarnings[1].4:=1;
			IF (nWarningArrayIndex<=5) THEN
				arrFaultMessage[nWarningArrayIndex+5]:='W005 - Filter #1 is Dirty';
				arrFaultWarningCurrent[nCurrent]:='W005 - Filter #1 is Dirty';
				nWarningArrayIndex:=nWarningArrayIndex+1;
				nCurrent:=nCurrent+1;
			END_IF
		END_IF

		IF nActiveWarnings[1].5=0 AND bMachineMode AND (fStartFeed=0) THEN
				nActiveWarnings[1].5:=1;
				IF (nWarningArrayIndex<=5) THEN
					arrFaultMessage[nWarningArrayIndex+5]:='W006a - Start Feedrate Must Be Nonzero';
					arrFaultWarningCurrent[nCurrent]:='W006a - Start Feedrate Must Be Nonzero';
					nWarningArrayIndex:=nWarningArrayIndex+1;
					nCurrent:=nCurrent+1;
				END_IF
		END_IF

		IF nActiveWarnings[1].6=0 AND bMachineMode AND (fFinishFeed=0) THEN
			nActiveWarnings[1].6:=1;
			IF (nWarningArrayIndex<=5) THEN
				arrFaultMessage[nWarningArrayIndex+5]:='W007 - Finish Feedrate Must Be Nonzero';
				arrFaultWarningCurrent[nCurrent]:='W007 - Finish Feedrate Must Be Nonzero';
				nWarningArrayIndex:=nWarningArrayIndex+1;
				nCurrent:=nCurrent+1;
			END_IF
		END_IF

		IF nActiveWarnings[1].7=0 AND NOT(bLubeLevel) AND bMCR THEN
			nActiveWarnings[1].7:=1;
			IF (nWarningArrayIndex<=5) THEN
				arrFaultMessage[nWarningArrayIndex+5]:='W008 - Lube Level Low';
				arrFaultWarningCurrent[nCurrent]:='W008 - Lube Level Low';
				nWarningArrayIndex:=nWarningArrayIndex+1;
				nCurrent:=nCurrent+1;
			END_IF
		ELSIF bLubeLevel AND nActiveWarnings[1].7=1 THEN
			IF FIND(arrFaultMessage[6], 'W008')>0 THEN
				arrFaultMessage[6]:=arrFaultMessage[7];
				arrFaultMessage[7]:=arrFaultMessage[8];
				arrFaultMessage[8]:=arrFaultMessage[9];
				arrFaultMessage[9]:=arrFaultMessage[10];
				arrFaultMessage[10]:='';
				nActiveWarnings[1].7:=0;
				nWarningArrayIndex:=nWarningArrayIndex-1;
			ELSIF FIND(arrFaultMessage[7], 'W008')>0 THEN
				arrFaultMessage[7]:=arrFaultMessage[8];
				arrFaultMessage[8]:=arrFaultMessage[9];
				arrFaultMessage[9]:=arrFaultMessage[10];
				arrFaultMessage[10]:='';
				nActiveWarnings[1].7:=0;
				nWarningArrayIndex:=nWarningArrayIndex-1;
			ELSIF FIND(arrFaultMessage[8], 'W008')>0 THEN
				arrFaultMessage[8]:=arrFaultMessage[9];
				arrFaultMessage[9]:=arrFaultMessage[10];
				arrFaultMessage[10]:='';
				nActiveWarnings[1].7:=0;
				nWarningArrayIndex:=nWarningArrayIndex-1;
			ELSIF FIND(arrFaultMessage[9], 'W008')>0 THEN
				arrFaultMessage[9]:=arrFaultMessage[10];
				arrFaultMessage[10]:='';
				nActiveWarnings[1].7:=0;
				nWarningArrayIndex:=nWarningArrayIndex-1;
			ELSIF FIND(arrFaultMessage[10], 'W008')>0 THEN
				arrFaultMessage[10]:='';
				nActiveWarnings[1].7:=0;
				nWarningArrayIndex:=nWarningArrayIndex-1;
			ELSE
				nActiveWarnings[1].7:=0;
				nWarningArrayIndex:=nWarningArrayIndex-1;
			END_IF
		END_IF

		IF nActiveWarnings[1].8=0 AND fbFilter2Timer.Q AND nDirtyCount2<5 THEN
			nDirtyCount2:=nDirtyCount2+1;
			nActiveWarnings[1].8:=1;
			IF (nWarningArrayIndex<=5) THEN
				arrFaultMessage[nWarningArrayIndex+5]:='W009 - Filter #2 is Dirty';
				arrFaultWarningCurrent[nCurrent]:='W009 - Filter #2 is Dirty';
				nWarningArrayIndex:=nWarningArrayIndex+1;
				nCurrent:=nCurrent+1;
			END_IF
		END_IF

		IF nActiveWarnings[1].9=0 AND fbFilter3Timer.Q AND nDirtyCount3<5 THEN
			nDirtyCount3:=nDirtyCount3+1;
			nActiveWarnings[1].9:=1;
			IF (nWarningArrayIndex<=5) THEN
				arrFaultMessage[nWarningArrayIndex+5]:='W010 - Filter #3 is Dirty';
				arrFaultWarningCurrent[nCurrent]:='W010 - Filter #3 is Dirty';
				nWarningArrayIndex:=nWarningArrayIndex+1;
				nCurrent:=nCurrent+1;
			END_IF
		END_IF

		IF nActiveWarnings[1].10=0 AND fbFilter4Timer.Q AND nDirtyCount4<5 THEN
			nDirtyCount4:=nDirtyCount4+1;
			nActiveWarnings[1].10:=1;
			IF (nWarningArrayIndex<=5) THEN
				arrFaultMessage[nWarningArrayIndex+5]:='W011 - Filter #4 is Dirty';
				arrFaultWarningCurrent[nCurrent]:='W011 - Filter #4 is Dirty';
				nWarningArrayIndex:=nWarningArrayIndex+1;
				nCurrent:=nCurrent+1;
			END_IF
		END_IF

		IF nActiveWarnings[1].11=0 AND bMCR AND NOT(bPneumaticSystemPressure) THEN
			nActiveWarnings[1].11:=1;
			IF (nWarningArrayIndex<=5) THEN
				arrFaultMessage[nWarningArrayIndex+5]:='W012 - Main Air Pressure Lost';
				arrFaultWarningCurrent[nCurrent]:='W012 - Main Air Pressure Lost';
				nWarningArrayIndex:=nWarningArrayIndex+1;
				nCurrent:=nCurrent+1;
			END_IF
		ELSIF bPneumaticSystemPressure AND nActiveWarnings[1].11 THEN
			IF FIND(arrFaultMessage[6], 'W012')>0 THEN
				arrFaultMessage[6]:=arrFaultMessage[7];
				arrFaultMessage[7]:=arrFaultMessage[8];
				arrFaultMessage[8]:=arrFaultMessage[9];
				arrFaultMessage[9]:=arrFaultMessage[10];
				arrFaultMessage[10]:='';
				nActiveWarnings[1].11:=0;
				nWarningArrayIndex:=nWarningArrayIndex-1;
			ELSIF FIND(arrFaultMessage[7], 'W012')>0 THEN
				arrFaultMessage[7]:=arrFaultMessage[8];
				arrFaultMessage[8]:=arrFaultMessage[9];
				arrFaultMessage[9]:=arrFaultMessage[10];
				arrFaultMessage[10]:='';
				nActiveWarnings[1].11:=0;
				nWarningArrayIndex:=nWarningArrayIndex-1;
			ELSIF FIND(arrFaultMessage[8], 'W012')>0 THEN
				arrFaultMessage[8]:=arrFaultMessage[9];
				arrFaultMessage[9]:=arrFaultMessage[10];
				arrFaultMessage[10]:='';
				nActiveWarnings[1].11:=0;
				nWarningArrayIndex:=nWarningArrayIndex-1;
			ELSIF FIND(arrFaultMessage[9], 'W012')>0 THEN
				arrFaultMessage[9]:=arrFaultMessage[10];
				arrFaultMessage[10]:='';
				nActiveWarnings[1].11:=0;
				nWarningArrayIndex:=nWarningArrayIndex-1;
			ELSIF FIND(arrFaultMessage[10], 'W012')>0 THEN
				arrFaultMessage[10]:='';
				nActiveWarnings[1].11:=0;
				nWarningArrayIndex:=nWarningArrayIndex-1;
			ELSE
				nActiveWarnings[1].11:=0;
				nWarningArrayIndex:=nWarningArrayIndex-1;
			END_IF
		END_IF

		IF nActiveWarnings[1].12=0 AND NOT(bProx311)
			AND (bMachineMode OR bEnterAutoModePB) AND NOT(bInCycle) THEN
			nActiveWarnings[1].12:=1;
			IF (nWarningArrayIndex<=5) THEN
				arrFaultMessage[nWarningArrayIndex+5]:='W013 - Tool Change Door Open Side B';
				arrFaultWarningCurrent[nCurrent]:='W013 - Tool Change Door Open Side B';
				nWarningArrayIndex:=nWarningArrayIndex+1;
				nCurrent:=nCurrent+1;
			END_IF
		ELSIF bProx311 AND nActiveWarnings[1].12 THEN
			IF FIND(arrFaultMessage[6], 'W013')>0 THEN
				arrFaultMessage[6]:=arrFaultMessage[7];
				arrFaultMessage[7]:=arrFaultMessage[8];
				arrFaultMessage[8]:=arrFaultMessage[9];
				arrFaultMessage[9]:=arrFaultMessage[10];
				arrFaultMessage[10]:='';
				nActiveWarnings[1].12:=0;
				nWarningArrayIndex:=nWarningArrayIndex-1;
			ELSIF FIND(arrFaultMessage[7], 'W013')>0 THEN
				arrFaultMessage[7]:=arrFaultMessage[8];
				arrFaultMessage[8]:=arrFaultMessage[9];
				arrFaultMessage[9]:=arrFaultMessage[10];
				arrFaultMessage[10]:='';
				nActiveWarnings[1].12:=0;
				nWarningArrayIndex:=nWarningArrayIndex-1;
			ELSIF FIND(arrFaultMessage[8], 'W013')>0 THEN
				arrFaultMessage[8]:=arrFaultMessage[9];
				arrFaultMessage[9]:=arrFaultMessage[10];
				arrFaultMessage[10]:='';
				nActiveWarnings[1].12:=0;
				nWarningArrayIndex:=nWarningArrayIndex-1;
			ELSIF FIND(arrFaultMessage[9], 'W013')>0 THEN
				arrFaultMessage[9]:=arrFaultMessage[10];
				arrFaultMessage[10]:='';
				nActiveWarnings[1].12:=0;
				nWarningArrayIndex:=nWarningArrayIndex-1;
			ELSIF FIND(arrFaultMessage[10], 'W013')>0 THEN
				arrFaultMessage[10]:='';
				nActiveWarnings[1].12:=0;
				nWarningArrayIndex:=nWarningArrayIndex-1;
			ELSE
				nActiveWarnings[1].12:=0;
				nWarningArrayIndex:=nWarningArrayIndex-1;
			END_IF
		END_IF

		IF nActiveWarnings[1].13=0 AND nModeError=Er_LoadPartMissing THEN
			nActiveWarnings[1].13:=1;
			nModeError:=Er_NoModeError;
			IF (nWarningArrayIndex<=5) THEN
				arrFaultMessage[nWarningArrayIndex+5]:='W014 - Load Side Missing Parts';
				arrFaultWarningCurrent[nCurrent]:='W014 - Load Side Missing Parts';
				nWarningArrayIndex:=nWarningArrayIndex+1;
				nCurrent:=nCurrent+1;
			END_IF
		END_IF

		IF nActiveWarnings[1].14=0 AND nModeError=Er_UnloadPartPresent THEN
			nActiveWarnings[1].14:=1;
			nModeError:=Er_NoModeError;
			IF (nWarningArrayIndex<=5) THEN
				arrFaultMessage[nWarningArrayIndex+5]:='W015 - Unload Side Remove Parts';
				arrFaultWarningCurrent[nCurrent]:='W015 - Unload Side Remove Parts';
				nWarningArrayIndex:=nWarningArrayIndex+1;
				nCurrent:=nCurrent+1;
			END_IF
		END_IF

		IF nActiveWarnings[1].15=0 AND nModeError=Er_TryingToLeaveAutoInCycle THEN
			nActiveWarnings[1].15:=1;
			nModeError:=Er_NoModeError;
			IF (nWarningArrayIndex<=5) THEN
				arrFaultMessage[nWarningArrayIndex+5]:='W016 - Can Not Exit Auto while in Cycle';
				arrFaultWarningCurrent[nCurrent]:='W016 - Can Not Exit Auto while in Cycle';
				nWarningArrayIndex:=nWarningArrayIndex+1;
				nCurrent:=nCurrent+1;
			END_IF
		END_IF

		IF nActiveWarnings[1].16=0 AND nModeError=Er_HydraulicPSOff THEN
			nActiveWarnings[1].16:=1;
			nModeError:=Er_NoModeError;
			IF (nWarningArrayIndex<=5) THEN
				arrFaultMessage[nWarningArrayIndex+5]:='W017 - Hydraulic Pressure Low';
				arrFaultWarningCurrent[nCurrent]:='W017 - Hydraulic Pressure Low';
				nWarningArrayIndex:=nWarningArrayIndex+1;
				nCurrent:=nCurrent+1;
			END_IF
		END_IF

		IF nActiveWarnings[1].17=0 AND nModeError=Er_XAxisNotHomed THEN
			nActiveWarnings[1].17:=1;
			nModeError:=Er_NoModeError;
			IF (nWarningArrayIndex<=5) THEN
				arrFaultMessage[nWarningArrayIndex+5]:='W018 - X Axis must be Homed';
				arrFaultWarningCurrent[nCurrent]:='W018 - X Axis must be Homed';
				nWarningArrayIndex:=nWarningArrayIndex+1;
				nCurrent:=nCurrent+1;
			END_IF
		END_IF

		IF nActiveWarnings[1].18=0 AND nModeError=Er_ZAAxisNotHomed THEN
			nActiveWarnings[1].18:=1;
			nModeError:=Er_NoModeError;
			IF (nWarningArrayIndex<=5) THEN
				arrFaultMessage[nWarningArrayIndex+5]:='W019 - ZA Axis must be Homed';
				arrFaultWarningCurrent[nCurrent]:='W019 - ZA Axis must be Homed';
				nWarningArrayIndex:=nWarningArrayIndex+1;
				nCurrent:=nCurrent+1;
			END_IF
		END_IF

		IF nActiveWarnings[1].19=0 AND nModeError=Er_WAAxisNotHomed THEN
			nActiveWarnings[1].19:=1;
			nModeError:=Er_NoModeError;
			IF (nWarningArrayIndex<=5) THEN
				arrFaultMessage[nWarningArrayIndex+5]:='W020 - WA Axis must be Homed';
				arrFaultWarningCurrent[nCurrent]:='W020 - WA Axis must be Homed';
				nWarningArrayIndex:=nWarningArrayIndex+1;
				nCurrent:=nCurrent+1;
			END_IF
		END_IF

		IF nActiveWarnings[1].20=0 AND nModeError=Er_ZBAxisNotHomed THEN
			nActiveWarnings[1].20:=1;
			nModeError:=Er_NoModeError;
			IF (nWarningArrayIndex<=5) THEN
				arrFaultMessage[nWarningArrayIndex+5]:='W021 - ZB Axis must be Homed';
				arrFaultWarningCurrent[nCurrent]:='W021 - ZB Axis must be Homed';
				nWarningArrayIndex:=nWarningArrayIndex+1;
				nCurrent:=nCurrent+1;
			END_IF
		END_IF

		IF nActiveWarnings[1].21=0 AND nModeError=Er_WBAxisNotHomed THEN
			nActiveWarnings[1].21:=1;
			nModeError:=Er_NoModeError;
			IF (nWarningArrayIndex<=5) THEN
				arrFaultMessage[nWarningArrayIndex+5]:='W022 - WB Axis must be Homed';
				arrFaultWarningCurrent[nCurrent]:='W022 - WB Axis must be Homed';
				nWarningArrayIndex:=nWarningArrayIndex+1;
				nCurrent:=nCurrent+1;
			END_IF
		END_IF

		IF nActiveWarnings[1].22=0 AND nModeError=Er_WANotRetracted THEN
			nActiveWarnings[1].22:=1;
			nModeError:=Er_NoModeError;
			IF (nWarningArrayIndex<=5) THEN
				arrFaultMessage[nWarningArrayIndex+5]:='W023 - Tailstock WA must be Retracted';
				arrFaultWarningCurrent[nCurrent]:='W022 - WB Axis must be Homed';
				nWarningArrayIndex:=nWarningArrayIndex+1;
				nCurrent:=nCurrent+1;
			END_IF
		END_IF

		IF nActiveWarnings[1].23=0 AND nModeError=Er_WBNotRetracted THEN
			nActiveWarnings[1].23:=1;
			nModeError:=Er_NoModeError;
			IF (nWarningArrayIndex<=5) THEN
				arrFaultMessage[nWarningArrayIndex+5]:='W024 - Tailstock WB must be Retracted';
				arrFaultWarningCurrent[nCurrent]:='W024 - Tailstock WB must be Retracted';
				nWarningArrayIndex:=nWarningArrayIndex+1;
				nCurrent:=nCurrent+1;
			END_IF
		END_IF

		IF nActiveWarnings[1].24=0 AND nModeError=Er_TransferNotAtLoad THEN
			nActiveWarnings[1].24:=1;
			nModeError:=Er_NoModeError;
			IF (nWarningArrayIndex<=5) THEN
				arrFaultMessage[nWarningArrayIndex+5]:='W025 - Transfer is not at Load Position';
				arrFaultWarningCurrent[nCurrent]:='W025 - Transfer is not at Load Position';
				nWarningArrayIndex:=nWarningArrayIndex+1;
				nCurrent:=nCurrent+1;
			END_IF
		END_IF

		IF nActiveWarnings[1].25=0 AND nModeError=Er_ACulletNotUnclamped THEN
			nActiveWarnings[1].25:=1;
			nModeError:=Er_NoModeError;
			IF (nWarningArrayIndex<=5) THEN
				arrFaultMessage[nWarningArrayIndex+5]:='W026 - Side A Collets Must Be Unclamped';
				arrFaultWarningCurrent[nCurrent]:='W026 - Side A Collets Must Be Unclamped';
				nWarningArrayIndex:=nWarningArrayIndex+1;
				nCurrent:=nCurrent+1;
			END_IF
		END_IF

		IF nActiveWarnings[1].26=0 AND nModeError=Er_BCulletNotUnclamped THEN
			nActiveWarnings[1].26:=1;
			nModeError:=Er_NoModeError;
			IF (nWarningArrayIndex<=5) THEN
				arrFaultMessage[nWarningArrayIndex+5]:='W027 - Side B Collets Must Be Unclamped';
				arrFaultWarningCurrent[nCurrent]:='W027 - Side B Collets Must Be Unclamped';
				nWarningArrayIndex:=nWarningArrayIndex+1;
				nCurrent:=nCurrent+1;
			END_IF
		END_IF

		IF nActiveWarnings[1].27=0 AND nModeError=Er_AEjectorsNotRetracted THEN
			nActiveWarnings[1].27:=1;
			nModeError:=Er_NoModeError;
			IF (nWarningArrayIndex<=5) THEN
				arrFaultMessage[nWarningArrayIndex+5]:='W028 - Side A Ejectors Not Retracted';
				arrFaultWarningCurrent[nCurrent]:='W028 - Side A Ejectors Not Retracted';
				nWarningArrayIndex:=nWarningArrayIndex+1;
				nCurrent:=nCurrent+1;
			END_IF
		END_IF

		IF nActiveWarnings[1].28=0 AND nModeError=Er_BEjectorsNotRetracted THEN
			nActiveWarnings[1].28:=1;
			nModeError:=Er_NoModeError;
			IF (nWarningArrayIndex<=5) THEN
				arrFaultMessage[nWarningArrayIndex+5]:='W029 - Side B Ejectors Not Retracted';
				arrFaultWarningCurrent[nCurrent]:='W029 - Side B Ejectors Not Retracted';
				nWarningArrayIndex:=nWarningArrayIndex+1;
				nCurrent:=nCurrent+1;
			END_IF
		END_IF

		IF nActiveWarnings[1].29=0 AND nModeError=Er_HPPumpOff THEN
			nActiveWarnings[1].29:=1;
			nModeError:=Er_NoModeError;
			IF (nWarningArrayIndex<=5) THEN
				arrFaultMessage[nWarningArrayIndex+5]:='W030 - Coolant System is OFF';
				arrFaultWarningCurrent[nCurrent]:='W030 - Coolant System is OFF';
				nWarningArrayIndex:=nWarningArrayIndex+1;
				nCurrent:=nCurrent+1;
			END_IF
		END_IF

		IF nActiveWarnings[1].30=0 AND bChipConveyorVFDFault THEN
			nActiveWarnings[1].30:=1;
			IF (nWarningArrayIndex<=5) THEN
				arrFaultMessage[nWarningArrayIndex+5]:='W031 - Chip Conveyor VFD Error';
				arrFaultWarningCurrent[nCurrent]:='W031 - Chip Conveyor VFD Error';
				nWarningArrayIndex:=nWarningArrayIndex+1;
				nCurrent:=nCurrent+1;
			END_IF
		ELSIF NOT(bMPGAOn) AND nActiveWarnings[1].30 THEN
			IF FIND(arrFaultMessage[6], 'W031')>0 THEN
				arrFaultMessage[6]:=arrFaultMessage[7];
				arrFaultMessage[7]:=arrFaultMessage[8];
				arrFaultMessage[8]:=arrFaultMessage[9];
				arrFaultMessage[9]:=arrFaultMessage[10];
				arrFaultMessage[10]:='';
				nActiveWarnings[1].30:=0;
				nWarningArrayIndex:=nWarningArrayIndex-1;
			ELSIF FIND(arrFaultMessage[7], 'W031')>0 THEN
				arrFaultMessage[7]:=arrFaultMessage[8];
				arrFaultMessage[8]:=arrFaultMessage[9];
				arrFaultMessage[9]:=arrFaultMessage[10];
				arrFaultMessage[10]:='';
				nActiveWarnings[1].30:=0;
				nWarningArrayIndex:=nWarningArrayIndex-1;
			ELSIF FIND(arrFaultMessage[8], 'W031')>0 THEN
				arrFaultMessage[8]:=arrFaultMessage[9];
				arrFaultMessage[9]:=arrFaultMessage[10];
				arrFaultMessage[10]:='';
				nActiveWarnings[1].30:=0;
				nWarningArrayIndex:=nWarningArrayIndex-1;
			ELSIF FIND(arrFaultMessage[9], 'W031')>0 THEN
				arrFaultMessage[9]:=arrFaultMessage[10];
				arrFaultMessage[10]:='';
				nActiveWarnings[1].30:=0;
				nWarningArrayIndex:=nWarningArrayIndex-1;
			ELSIF FIND(arrFaultMessage[10], 'W031')>0 THEN
				arrFaultMessage[10]:='';
				nActiveWarnings[1].30:=0;
				nWarningArrayIndex:=nWarningArrayIndex-1;
			ELSE
				nActiveWarnings[1].30:=0;
				nWarningArrayIndex:=nWarningArrayIndex-1;
			END_IF
		END_IF

		IF nActiveWarnings[1].31=0 AND bHydraulicTemperature AND
			(bHydraulicUnitOn AND fbHydraulicSystemOnTON.Q)
		THEN
			nActiveWarnings[1].31:=1;
			IF (nWarningArrayIndex<=5) THEN
				arrFaultMessage[nWarningArrayIndex+5]:='W032 - Hydraulic Fluid Temperature High Alarm';
				arrFaultWarningCurrent[nCurrent]:='W032 - Hydraulic Fluid Temperature High Alarm';
				nWarningArrayIndex:=nWarningArrayIndex+1;
				nCurrent:=nCurrent+1;
			END_IF
		END_IF

		IF nActiveWarnings[2].0=0 AND fbLubePressureTON.Q THEN
			nActiveWarnings[2].0:=1;
			IF (nWarningArrayIndex<=5) THEN
				arrFaultMessage[nWarningArrayIndex+5]:='W033 - Lube Pressure Lost';
				arrFaultWarningCurrent[nCurrent]:='W033 - Lube Pressure Lost';
				nWarningArrayIndex:=nWarningArrayIndex+1;
				nCurrent:=nCurrent+1;
			END_IF
		END_IF

		IF nActiveWarnings[2].1=0 AND fbHydraulicFluidLowTON.Q THEN
			nActiveWarnings[2].1:=1;
			IF (nWarningArrayIndex<=5) THEN
				arrFaultMessage[nWarningArrayIndex+5]:='W034 - Hydraulic Unit Fluid Level Low';
				arrFaultWarningCurrent[nCurrent]:='W034 - Hydraulic Unit Fluid Level Low';
				nWarningArrayIndex:=nWarningArrayIndex+1;
				nCurrent:=nCurrent+1;
			END_IF
		END_IF

		IF nActiveWarnings[2].2=0 AND MAIN.fbChipConveyorMotorControl.bError THEN
			nActiveWarnings[2].2:=1;
			IF (nWarningArrayIndex<=5) THEN
				arrFaultMessage[nWarningArrayIndex+5]:='W035 - Chip Conveyor MS-3 Failure';
				arrFaultWarningCurrent[nCurrent]:='W035 - Chip Conveyor MS-3 Failure';
				nWarningArrayIndex:=nWarningArrayIndex+1;
				nCurrent:=nCurrent+1;
			END_IF
		END_IF

		IF nActiveWarnings[2].3=0 AND bMachineMode THEN
			IF  fFinishDepth=0 THEN
				nActiveWarnings[2].3:=1;
				IF (nWarningArrayIndex<=5) THEN
					arrFaultMessage[nWarningArrayIndex+5]:='W036a - Finish Depth Must Be Nonzero';
					arrFaultWarningCurrent[nCurrent]:='W036a - Finish Depth Must Be Nonzero';
					nWarningArrayIndex:=nWarningArrayIndex+1;
					nCurrent:=nCurrent+1;
				END_IF
			ELSIF fStartDepth < fFinishDepth THEN
				nActiveWarnings[2].3:=1;
				IF (nWarningArrayIndex<=5) THEN
					arrFaultMessage[nWarningArrayIndex+5]:='W036b - Check Start Depth';
					arrFaultWarningCurrent[nCurrent]:='W036b - Check Start Depth';
					nWarningArrayIndex:=nWarningArrayIndex+1;
					nCurrent:=nCurrent+1;
				END_IF
			END_IF
		END_IF

		(* Coolant Pressure Warning Side A in Setup Mode *)
		IF nActiveWarnings[2].4=0 AND fbLowPressureFaultADelay.Q
				AND NOT bMachineMode
			THEN
			nActiveWarnings[2].4:=1;
			IF (nWarningArrayIndex<=5) THEN
				arrFaultMessage[nWarningArrayIndex+5]:='W037 - Coolant Pressure Low - Side A';
				arrFaultWarningCurrent[nCurrent]:='W037 - Coolant Pressure Low - Side A';
				nWarningArrayIndex:=nWarningArrayIndex+1;
				nCurrent:=nCurrent+1;
			END_IF
		ELSIF  nActiveWarnings[2].4 AND (NOT(bACoolantSolenoid) OR bACoolantPressure) THEN
			IF FIND(arrFaultMessage[6], 'W037')>0 THEN
				arrFaultMessage[6]:=arrFaultMessage[7];
				arrFaultMessage[7]:=arrFaultMessage[8];
				arrFaultMessage[8]:=arrFaultMessage[9];
				arrFaultMessage[9]:=arrFaultMessage[10];
				arrFaultMessage[10]:='';
				nActiveWarnings[2].4:=0;
				nWarningArrayIndex:=nWarningArrayIndex-1;
			ELSIF FIND(arrFaultMessage[7], 'W037')>0 THEN
				arrFaultMessage[7]:=arrFaultMessage[8];
				arrFaultMessage[8]:=arrFaultMessage[9];
				arrFaultMessage[9]:=arrFaultMessage[10];
				arrFaultMessage[10]:='';
				nActiveWarnings[2].4:=0;
				nWarningArrayIndex:=nWarningArrayIndex-1;
			ELSIF FIND(arrFaultMessage[8], 'W037')>0 THEN
				arrFaultMessage[8]:=arrFaultMessage[9];
				arrFaultMessage[9]:=arrFaultMessage[10];
				arrFaultMessage[10]:='';
				nActiveWarnings[2].4:=0;
				nWarningArrayIndex:=nWarningArrayIndex-1;
			ELSIF FIND(arrFaultMessage[9], 'W037')>0 THEN
				arrFaultMessage[9]:=arrFaultMessage[10];
				arrFaultMessage[10]:='';
				nActiveWarnings[2].4:=0;
				nWarningArrayIndex:=nWarningArrayIndex-1;
			ELSIF FIND(arrFaultMessage[10], 'W037')>0 THEN
				arrFaultMessage[10]:='';
				nActiveWarnings[2].4:=0;
				nWarningArrayIndex:=nWarningArrayIndex-1;
			ELSE
				nActiveWarnings[2].4:=0;
				nWarningArrayIndex:=nWarningArrayIndex-1;
			END_IF
		END_IF

		(* Coolant Pressure Warning Side B in Setup Mode *)
		IF nActiveWarnings[2].5=0 AND fbLowPressureFaultBDelay.Q
				AND NOT bMachineMode
			THEN
			nActiveWarnings[2].5:=1;
			IF (nWarningArrayIndex<=5) THEN
				arrFaultMessage[nWarningArrayIndex+5]:='W038 - Coolant Pressure Low - Side B';
				arrFaultWarningCurrent[nCurrent]:='W038 - Coolant Pressure Low - Side B';
				nWarningArrayIndex:=nWarningArrayIndex+1;
				nCurrent:=nCurrent+1;
			END_IF
		ELSIF  nActiveWarnings[2].5 AND (NOT(bBCoolantSolenoid) OR bBCoolantPressure) THEN
			IF FIND(arrFaultMessage[6], 'W038')>0 THEN
				arrFaultMessage[6]:=arrFaultMessage[7];
				arrFaultMessage[7]:=arrFaultMessage[8];
				arrFaultMessage[8]:=arrFaultMessage[9];
				arrFaultMessage[9]:=arrFaultMessage[10];
				arrFaultMessage[10]:='';
				nActiveWarnings[2].5:=0;
				nWarningArrayIndex:=nWarningArrayIndex-1;
			ELSIF FIND(arrFaultMessage[7], 'W038')>0 THEN
				arrFaultMessage[7]:=arrFaultMessage[8];
				arrFaultMessage[8]:=arrFaultMessage[9];
				arrFaultMessage[9]:=arrFaultMessage[10];
				arrFaultMessage[10]:='';
				nActiveWarnings[2].5:=0;
				nWarningArrayIndex:=nWarningArrayIndex-1;
			ELSIF FIND(arrFaultMessage[8], 'W038')>0 THEN
				arrFaultMessage[8]:=arrFaultMessage[9];
				arrFaultMessage[9]:=arrFaultMessage[10];
				arrFaultMessage[10]:='';
				nActiveWarnings[2].5:=0;
				nWarningArrayIndex:=nWarningArrayIndex-1;
			ELSIF FIND(arrFaultMessage[9], 'W038')>0 THEN
				arrFaultMessage[9]:=arrFaultMessage[10];
				arrFaultMessage[10]:='';
				nActiveWarnings[2].5:=0;
				nWarningArrayIndex:=nWarningArrayIndex-1;
			ELSIF FIND(arrFaultMessage[10], 'W038')>0 THEN
				arrFaultMessage[10]:='';
				nActiveWarnings[2].5:=0;
				nWarningArrayIndex:=nWarningArrayIndex-1;
			ELSE
				nActiveWarnings[2].5:=0;
				nWarningArrayIndex:=nWarningArrayIndex-1;
			END_IF
		END_IF

(* SPARES *)

		(* MPGA Axis Selected *)
		bMPGAOn:=(bWAAxisSelected OR bXAAxisSelected OR bYAAxisSelected OR bZAAxisSelected);
		IF nActiveWarnings[2].12=0 AND (bMachineMode OR bEnterAutoModePB) AND
			bMPGAON AND NOT(bInCycle) THEN
			nActiveWarnings[2].12:=1;
			IF (nWarningArrayIndex<=5) THEN
				arrFaultMessage[nWarningArrayIndex+5]:='W130 - MPG A Must Be Off';
				arrFaultWarningCurrent[nCurrent]:='W130 - MPG A Must Be Off';
				nWarningArrayIndex:=nWarningArrayIndex+1;
				nCurrent:=nCurrent+1;
			END_IF
		ELSIF NOT(bMPGAOn) AND nActiveWarnings[2].12 THEN
			IF FIND(arrFaultMessage[6], 'W130')>0 THEN
				arrFaultMessage[6]:=arrFaultMessage[7];
				arrFaultMessage[7]:=arrFaultMessage[8];
				arrFaultMessage[8]:=arrFaultMessage[9];
				arrFaultMessage[9]:=arrFaultMessage[10];
				arrFaultMessage[10]:='';
				nActiveWarnings[2].12:=0;
				nWarningArrayIndex:=nWarningArrayIndex-1;
			ELSIF FIND(arrFaultMessage[7], 'W130')>0 THEN
				arrFaultMessage[7]:=arrFaultMessage[8];
				arrFaultMessage[8]:=arrFaultMessage[9];
				arrFaultMessage[9]:=arrFaultMessage[10];
				arrFaultMessage[10]:='';
				nActiveWarnings[2].12:=0;
				nWarningArrayIndex:=nWarningArrayIndex-1;
			ELSIF FIND(arrFaultMessage[8], 'W130')>0 THEN
				arrFaultMessage[8]:=arrFaultMessage[9];
				arrFaultMessage[9]:=arrFaultMessage[10];
				arrFaultMessage[10]:='';
				nActiveWarnings[2].12:=0;
				nWarningArrayIndex:=nWarningArrayIndex-1;
			ELSIF FIND(arrFaultMessage[9], 'W130')>0 THEN
				arrFaultMessage[9]:=arrFaultMessage[10];
				arrFaultMessage[10]:='';
				nActiveWarnings[2].12:=0;
				nWarningArrayIndex:=nWarningArrayIndex-1;
			ELSIF FIND(arrFaultMessage[10], 'W130')>0 THEN
				arrFaultMessage[10]:='';
				nActiveWarnings[2].12:=0;
				nWarningArrayIndex:=nWarningArrayIndex-1;
			ELSE
				nActiveWarnings[2].12:=0;
				nWarningArrayIndex:=nWarningArrayIndex-1;
			END_IF
		END_IF

		(* MPGB Axis Selected *)
		bMPGBOn:=(bWBAxisSelected OR bXBAxisSelected OR bYBAxisSelected OR bZBAxisSelected);
		IF nActiveWarnings[2].13=0 AND (bMachineMode OR bEnterAutoModePB) AND
			bMPGBON AND NOT(bInCycle) THEN
			nActiveWarnings[2].13:=1;
			IF (nWarningArrayIndex<=5) THEN
				arrFaultMessage[nWarningArrayIndex+5]:='W131 - MPG B Must Be Off';
				arrFaultWarningCurrent[nCurrent]:='W131 - MPG B Must Be Off';
				nWarningArrayIndex:=nWarningArrayIndex+1;
				nCurrent:=nCurrent+1;
			END_IF
		ELSIF NOT(bMPGAOn) AND nActiveWarnings[2].12 THEN
			IF FIND(arrFaultMessage[6], 'W131')>0 THEN
				arrFaultMessage[6]:=arrFaultMessage[7];
				arrFaultMessage[7]:=arrFaultMessage[8];
				arrFaultMessage[8]:=arrFaultMessage[9];
				arrFaultMessage[9]:=arrFaultMessage[10];
				arrFaultMessage[10]:='';
				nActiveWarnings[2].13:=0;
				nWarningArrayIndex:=nWarningArrayIndex-1;
			ELSIF FIND(arrFaultMessage[7], 'W131')>0 THEN
				arrFaultMessage[7]:=arrFaultMessage[8];
				arrFaultMessage[8]:=arrFaultMessage[9];
				arrFaultMessage[9]:=arrFaultMessage[10];
				arrFaultMessage[10]:='';
				nActiveWarnings[2].13:=0;
				nWarningArrayIndex:=nWarningArrayIndex-1;
			ELSIF FIND(arrFaultMessage[8], 'W131')>0 THEN
				arrFaultMessage[8]:=arrFaultMessage[9];
				arrFaultMessage[9]:=arrFaultMessage[10];
				arrFaultMessage[10]:='';
				nActiveWarnings[2].13:=0;
				nWarningArrayIndex:=nWarningArrayIndex-1;
			ELSIF FIND(arrFaultMessage[9], 'W131')>0 THEN
				arrFaultMessage[9]:=arrFaultMessage[10];
				arrFaultMessage[10]:='';
				nActiveWarnings[2].13:=0;
				nWarningArrayIndex:=nWarningArrayIndex-1;
			ELSIF FIND(arrFaultMessage[10], 'W131')>0 THEN
				arrFaultMessage[10]:='';
				nActiveWarnings[2].13:=0;
				nWarningArrayIndex:=nWarningArrayIndex-1;
			ELSE
				nActiveWarnings[2].13:=0;
				nWarningArrayIndex:=nWarningArrayIndex-1;
			END_IF
		END_IF

		(***** TRANSFER WARNINGS ****
		The text of the Warning comes from the the TransferCycle Action of the P_TransferControl (PGM). 
			We assign the 100 series to the warnings by concating a W1 to the beginning of the text.  
			This allows us to assign the Warning series of numbers in an effort to make it more modular.  
			You must go to the function block to see the rest of the number and the description text of the fault. f
			Generally this is at the bottom of the function block or program section. 
			ErrorID < 50 is a WARNING and ErrorID >= 50 are Faults
			If this is reused in a different machine we want to make sure we assign the appropriate #series to the warnings.  *)
		IF  nActiveWarnings[2].14=0  AND bTransferError  AND nTransferErrorID < 50THEN
			nActiveWarnings[2].14:=1;
			IF (nWarningArrayIndex<=5) THEN
				arrFaultMessage[nWarningArrayIndex+5]:=CONCAT('W1',sTransferErrorText);
				arrFaultWarningCurrent[nCurrent]:=CONCAT('W1',sTransferErrorText);
				nWarningArrayIndex:=nWarningArrayIndex+1;
				nCurrent:=nCurrent+1;
			END_IF
		END_IF

		IF nActiveWarnings[4].0=0 AND bLoadSideNotSelected THEN
			bLoadSideNotSelected:=FALSE;
			nActiveWarnings[4].0:=1;
			IF (nWarningArrayIndex<=5) THEN
				arrFaultMessage[nWarningArrayIndex+5]:='W??? - Load Side not selected - Call Maintenance';
				arrFaultWarningCurrent[nCurrent]:='W??? - Load Side not selected - Call Maintenance';;
				nWarningArrayIndex:=nWarningArrayIndex+1;
				nCurrent:=nCurrent+1;
			END_IF
		END_IF



		(* Did we have any faults? *)
		IF nActiveFaults[1]>0
		OR nActiveFaults[2]>0
		OR nActiveFaults[3]>0
		OR nActiveFaults[4]>0 THEN
			bMachineFault:=TRUE;
		END_IF
		(* Did we have any Warning? *)
		IF nActiveWarnings[1]>0
		OR nActiveWarnings[2]>0
		OR nActiveWarnings[3]>0
		OR nActiveWarnings[4]>0 THEN
			bMachineWarning:=TRUE;
		ELSE
			bMachineWarning:=FALSE;
		END_IF
		(* If so then we go to state 1 to wait for a Reset *)
		IF bMachineFault OR bMachineWarning THEN
			nFaultState:=nFaultState+1;
			(* Special condition withing the first 40 seconds of Master Start
				check for servo faults to trigger an Internal Fault Reset *)
			IF bMCR AND NOT  fbMCRJustOnTON.Q THEN
				IF bSideAEnabled AND ( stZAAxis.NcToPlc.StateDWord.31 OR
					stWAAxis.NcToPlc.StateDWord.31)
				THEN
					bAFaultResetInternal:=TRUE;
				END_IF
				IF bSideBEnabled AND (stZBAxis.NcToPlc.StateDWord.31 OR
					stWBAxis.NcToPlc.StateDWord.31)
				THEN
					bBFaultResetInternal:=TRUE;
				END_IF
				IF stUAxis.NcToPlc.StateDWord.31 THEN
					(* Just need to trigger a reset, so either side would do *)
					bAFaultResetInternal:=TRUE;
				END_IF
			END_IF
		(* When the Internal Resets are on and we do not have any faults we want to turn it off *)
		ELSIF fbInternalResetTON.Q THEN
			bAFaultResetInternal:=FALSE;
			bBFaultResetInternal:=FALSE;
		END_IF

	(* If we get a fault reset reset requested by a push button or internal request then we check the drives for faults .
	  If a drive has a fault then we set the bit to reset that drive.  The bit will be reset in the servo control section, 
		so we want to wait for it before we move on.
	  Once we no longer have any of the drives requiring a reset, then we jump to step 2. 
	  If we do not get a reset request or a drive reset then we go back and check for more faults. *)

	1:	(* Wait for Fault Resets *)

		(* When Fault Reset Requested we check to see if the drives are resetting *)
		IF bFaultResetRequested THEN
			(* The Drive Resets are cleared by the servo control sections *)
			IF NOT(bZWADriveResetRequest OR bZWBDriveResetRequest OR bUDriveResetRequest) OR
				(* Timer does not allow to get stuck in this step *)
				fbFaultResetWatchdog.Q
			 THEN
				bFaultResetRequested:=FALSE;
				nFaultState:=nFaultState+1;
			END_IF

		(* If Fault Reset PB's or internal reset then turn on reset requested *)
		ELSIF bFaultResetPB OR fbCommonFautlResetTON.Q OR
			bAFaultResetInternal OR bBFaultResetInternal
		THEN
			bFaultResetRequested:=TRUE;

			(* Do A reset of the Servo Drives if they are faulted, then we need to do a MCReset for the same drives *)

			(* Do a FB_SoEReset of the Drive when one of the Servo Axis has the Fault State bit set *)
			IF bSideAEnabled AND ( stZAAxis.NcToPlc.StateDWord.31 OR stWAAxis.NcToPlc.StateDWord.31) THEN
				bZWADriveResetRequest:=TRUE;
			END_IF
			IF bSideBEnabled AND (stZBAxis.NcToPlc.StateDWord.31 OR stWBAxis.NcToPlc.StateDWord.31) THEN
				bZWBDriveResetRequest:=TRUE;
			END_IF
			IF stUAxis.NcToPlc.StateDWord.31THEN
				bUDriveResetRequest:=TRUE;
			END_IF
			(* Reset the MPG if it is faulted *)
			IF stAxisMPG_A.NcToPlc.StateDWord.31 THEN
				bMPGA_MCResetRequest:=TRUE;
			END_IF
			IF stAxisMPG_B.NcToPlc.StateDWord.31 THEN
				bMPGB_MCResetRequest:=TRUE;
			END_IF

		(* Go back and check for more faults if no Reset action was requested *)
		ELSE
			nFaultState:=nFaultState-1;
		END_IF


	2:	(* Take Action on the Requested Fault *)
		(* Clear the Fault Display Messages and the Active Faults/Warnings *)
		arrFaultMessage[1]:='';
		arrFaultMessage[2]:='';
		arrFaultMessage[3]:='';
		arrFaultMessage[4]:='';
		arrFaultMessage[5]:='';
		arrFaultMessage[6]:='';
		arrFaultMessage[7]:='';
		arrFaultMessage[8]:='';
		arrFaultMessage[9]:='';
		arrFaultMessage[10]:='';
		nFaultArrayIndex:=1;
		nWarningArrayIndex:=1;
		nActiveFaults[1]:=0;
		nActiveFaults[2]:=0;
		nActiveFaults[3]:=0;
		nActiveFaults[4]:=0;
		nActiveWarnings[1]:=0;
		nActiveWarnings[2]:=0;
		nActiveWarnings[3]:=0;
		nActiveWarnings[4]:=0;
		bMachineFault:=FALSE;
		bMachineWarning:=FALSE;
		bFaultHistoryFileError:=FALSE;

		(* Reset the Filter Timers *)
		IF fbFilter1Timer.Q THEN
			bFilter1Timer:=FALSE;
		END_IF
		IF fbFilter2Timer.Q THEN
			bFilter2Timer:=FALSE;
		END_IF
		IF fbFilter3Timer.Q THEN
			bFilter3Timer:=FALSE;
		END_IF
		IF fbFilter4Timer.Q THEN
			bFilter4Timer:=FALSE;
		END_IF

		(* When the PB is Released then we jump out of this state or
			if it is internal reset we reset and jump out *)
		IF NOT(bFaultResetPB OR fbCommonFautlResetTON.Q) OR (* put two into one Not ored toghether *)
			bAFaultResetInternal OR bBFaultResetInternal
		THEN
			bAFaultResetInternal:=FALSE;
			bBFaultResetInternal:=FALSE;
			nFaultState:=0;
		END_IF

END_CASE

(* When the Internal Fault Reset has been on for a while without a bMachineFault we trigger a reset *)
fbInternalResetTON(IN:= (bAFaultResetInternal OR bBFaultResetInternal)
	AND NOT bMachineFault, PT:=t#250ms);
(* The Servo will sometimes fault and need to be reset withing 30 seconds of the MCR being pulled in *)
fbMCRJustOnTON(IN:=bMCR, PT:=t#40s);

(* When we have a fault we need to write it to fault history *)
IF nCurrent>nUnStored THEN
	(* This will take the number of nCurrent Scans to store current faults to history *)
	CASE nHistoryStep OF
	1:	(*	Copy nFaultHistory[1-79] to nFaultHistoryTemp[2-80]	*)
		IF MEMCPY(
			ADR(arrFaultHistoryTemp[2]),
			ADR(arrFaultHistory[1]),
			SIZEOF(arrFaultHistory)-SIZEOF(arrFaultHistory[1])
		) <> 0 THEN (* Returneing a Zero meanse Error*)
			nHistoryStep:=nHistoryStep+1;
		END_IF

	2:	(*	Copy current Fault/Waring into nFaultHistoryTemp[1]	*)
		IF MEMCPY(
			ADR(arrFaultHistoryTemp[1]),
			ADR(arrFaultWarningCurrent[nUnStored MOD 8]),
			SIZEOF(arrFaultHistoryTemp[1])
		) <> 0 THEN
			nHistoryStep:=nHistoryStep+1;
		END_IF

	3:	(*	Copy nFaultHistoryTemp to nFaultHistory	*)
		IF MEMCPY(
			ADR(arrFaultHistory[1]),
			ADR(arrFaultHistoryTemp[1]),
			SIZEOF(arrFaultHistory)
		) <> 0 THEN
			nHistoryStep:=1;
			(*	Increment nUnStored	*)
			nUnStored:=nUnStored+1;
		END_IF

	END_CASE

ELSIF nCurrent=nUnStored THEN
	nCurrent:=0;
	nUnStored:=0;
END_IF

(* Coolant Temp Monitoring *)
fCoolantTempDisplay:=(nCoolantTemp/10.0);
IF fCoolantTempDisplay>=43.33 THEN
	bCoolantTempFault:=TRUE;
ELSIF fCoolantTempDisplay>=40.55 THEN
	bCoolantTempWarning:=TRUE;
	bCoolantTempFault:=FALSE;
ELSE
	bCoolantTempFault:=FALSE;
	bCoolantTempWarning:=FALSE;
END_IF

fbFaultResetWatchdog(IN:=bFaultResetRequested, PT:=t#5s);
END_PROGRAM

(* POU Programs/P_MPGControl, ST *)
PROGRAM P_MPGControl
VAR

	fbMPGAAxisEnable: MC_Power;
	bMPGAAxisEnable : BOOL := FALSE;

	fbMPGBAxisEnable: MC_Power;
	bMPGBAxisEnable : BOOL := FALSE;

	fbMPGUAOn: R_TRIG;
	fbMPGYAOn: R_TRIG;
	fbMPGZAOn: R_TRIG;
	fbMPGWAOn: R_TRIG;

	fbMPGXBOn: R_TRIG;
	fbMPGYBOn: R_TRIG;
	fbMPGZBOn: R_TRIG;
	fbMPGWBOn: R_TRIG;

	fbAAxisSelectDelay: TON;				(* Side A MPG Axis Selected Delay Timer *)

	fbBAxisSelectDelay: TON;				(* Side B MPG Axis Selected Delay Timer *)

	fbMPGUAAxisGearIn: MC_GearInDyn;
	bMPGUAAxisGearIn : BOOL;
	fbMPGUAAxisGearOut : MC_GearOut;
	bMPGUAAxisGearOut : BOOL;

	fbMPGZAAxisGearIn : MC_GearInDyn;
	bMPGZAAxisGearIn : BOOL;
	fbMPGZAAxisGearOut : MC_GearOut;
	bMPGZAAxisGearOut : BOOL;

	fbMPGWAAxisGearIn : MC_GearInDyn;
	bMPGWAAxisGearIn : BOOL;
	fbMPGWAAxisGearOut : MC_GearOut;
	bMPGWAAxisGearOut : BOOL;

	fbMPGXBAxisGearIn: MC_GearInDyn;
	bMPGXBAxisGearIn : BOOL;
	fbMPGXBAxisGearOut : MC_GearOut;
	bMPGXBAxisGearOut : BOOL;

	fbMPGZBAxisGearIn : MC_GearInDyn;
	bMPGZBAxisGearIn : BOOL;
	fbMPGZBAxisGearOut : MC_GearOut;
	bMPGZBAxisGearOut : BOOL;

	fbMPGWBAxisGearIn : MC_GearInDyn;
	bMPGWBAxisGearIn : BOOL;
	fbMPGWBAxisGearOut : MC_GearOut;
	bMPGWBAxisGearOut : BOOL;

	MPG_A_Rate: INT := 1;		(*Side A MPG Rate*)
	MPG_B_Rate: INT := 1;		(*Side B MPG Rate*)

	MPGMode: INT := 0;		(*MPG State Mode Counter*)
	nMPG_A_State: INT := 0;		(*MPG Side A State Counter*)
	nMPG_B_State: INT := 0;		(*MPG Side A State Counter*)

	nMPGA_ErrorID : UDINT := 0;
	fGearRatioA: LREAL := 0.1;		(*Gear Ratio Input to the Gear In FB*)
	nMPGB_ErrorID : UDINT := 0;
	fGearRatioB: LREAL := 0.1;		(*Gear Ratio Input to the Gear In FB*)

	fbMPGWatchdog : TON;			(* Watchdog Timer for MPG A Control *)
	bMPGWatchdog : BOOL := FALSE;	(* Watchdog Timer TRigger for MPG A *)
	fbMPGBWatchdog : TON;			(* Watchdog Timer for MPG  B Control *)
	bMPGBWatchdog : BOOL := FALSE;	(* Watchdog Timer TRigger for MPG B *)
END_VAR
(* When the MCC_S comes in Enable the MPG's *)
bMPGAAxisEnable := bMCC_SConfirm;
bMPGBAxisEnable := bMCC_SConfirm;

(* Only Available if Manual Mode and the MCC_S pulled in *)
IF bMCC_SConfirm AND NOT bMachineMode THEN
	CASE MPGMode OF
		0: (* Check if an Axis is selected *)
			IF bMachineFault THEN	(* Fault so stay in this step *)
				MPGMode := 0;
				nMPG_A_State:=0;
				(* Do not really need to Gear Out at this point, but this is what the Eaton program did *)
				bMPGUAAxisGearOut := TRUE;
				bMPGZAAxisGearOut := TRUE;
				bMPGWAAxisGearOut := TRUE;
				bMPGXBAxisGearOut := TRUE;
				bMPGZBAxisGearOut := TRUE;
				bMPGWBAxisGearOut := TRUE;
			ELSIF fbMPGUAOn.Q THEN
				bMPGUAAxisGearIn := FALSE;
				bMPGUAAxisGearOut := FALSE;
				MPGMode := 1;
			ELSIF fbMPGZAOn.Q THEN
				bMPGZAAxisGearIn := FALSE;
				bMPGZAAxisGearOut := FALSE;
				MPGMode := 3;
			ELSIF fbMPGWAOn.Q THEN
				bMPGWAAxisGearIn := FALSE;
				bMPGWAAxisGearOut := FALSE;
				MPGMode := 4;
			ELSIF fbMPGXBOn.Q THEN
				bMPGXBAxisGearIn := FALSE;
				bMPGXBAxisGearOut := FALSE;
				MPGMode := 5;
			ELSIF fbMPGZBOn.Q THEN
				bMPGZBAxisGearIn := FALSE;
				bMPGZBAxisGearOut := FALSE;
				MPGMode := 7;
			ELSIF fbMPGWBOn.Q THEN
				bMPGWBAxisGearIn := FALSE;
				bMPGWBAxisGearOut := FALSE;
				MPGMode := 8;
			END_IF

		1: (* U Axis Selected *)
			CASE nMPG_A_State OF
			0:	(* INIT *)
				IF NOT bXAAxisSelected THEN
					MPGMode := 0;
				ELSE
					nMPG_A_State := nMPG_A_State + 1;
				END_IF

			1:	(* Request Gear In *)
				IF bMPGUAAxisGearIn AND fbMPGUAAxisGearIn.InGear THEN
					nMPG_A_State:=nMPG_A_State+1;
				ELSIF bMPGUAAxisGearIn AND fbMPGUAAxisGearIn.Error THEN
					bMPGUAAxisGearIn := FALSE;
					nMPGA_ErrorID := fbMPGUAAxisGearIn.ErrorID;
					nMPG_A_State := 5;
				ELSE
					bMPGUAAxisGearIn:=TRUE;
				END_IF

			2:	(* Wait for Axis Selector Change or end if a Fault Occurs *)
				IF NOT(bXAAxisSelected) OR bMachineFault THEN
					bMPGUAAxisGearIn:=FALSE;
					nMPG_A_State:=nMPG_A_State+1;
				END_IF

			3:	(* Request Gear Out *)
				IF bMPGUAAxisGearOut AND fbMPGUAAxisGearOut.Done AND NOT(fbMPGUAAxisGearOut.Error) THEN
					bMPGUAAxisGearOut:=FALSE;
					nMPG_A_State := nMPG_A_State+1;
				ELSIF bMPGUAAxisGearOut AND fbMPGUAAxisGearOut.Error THEN
					bMPGUAAxisGearOut:=FALSE;
					nMPGA_ErrorID := fbMPGUAAxisGearOut.ErrorID;
					nMPG_A_State:=4;
				ELSE
					bMPGUAAxisGearOut:=TRUE;
				END_IF

			4:	(* Request Axis Stop *)
				IF bUStop AND fbUAxisStop.Done	AND NOT(fbUAxisStop.Error) THEN
					bUStop:=FALSE;
					nMPG_A_State:=nMPG_A_State+1;
				ELSIF bUStop AND fbUAxisStop.Error THEN
					bUStop:=FALSE;
					nMPG_A_State:=5;
				ELSE
					bUStop:=TRUE;
				END_IF

			5:	(* Fault/Clean Up State *)
				bUStop:=FALSE;
				bMPGUAAxisGearIn:=FALSE;
				bMPGUAAxisGearOut:=FALSE;
				IF NOT(bXAAxisSelected) THEN
					nMPG_A_State:=0;
					MPGMode := 0;
				END_IF
			END_CASE	(* U *)

		3: (* ZA Axis Selected *)
			CASE nMPG_A_State OF
			0:	(* INIT *)
				IF NOT bZAAxisSelected THEN
					MPGMode := 0;
				ELSE
					nMPG_A_State := nMPG_A_State + 1;
				END_IF

			1:	(* Request Gear In *)
				IF bMPGZAAxisGearIn AND fbMPGZAAxisGearIn.InGear THEN
					nMPG_A_State:=nMPG_A_State+1;
				ELSIF bMPGZAAxisGearIn AND fbMPGZAAxisGearIn.Error THEN
					bMPGZAAxisGearIn := FALSE;
					nMPGA_ErrorID := fbMPGZAAxisGearIn.ErrorID;
					nMPG_A_State := 5;
				ELSE
					bMPGZAAxisGearIn:=TRUE;
				END_IF

			2:	(* Wait for Axis Selector Change or end if a Fault Occurs *)
				IF NOT(bZAAxisSelected) OR bMachineFault THEN
					bMPGZAAxisGearIn:=FALSE;
					nMPG_A_State:=nMPG_A_State+1;
				END_IF

			3:	(* Request Gear Out *)
				IF bMPGZAAxisGearOut AND fbMPGZAAxisGearOut.Done AND NOT(fbMPGZAAxisGearOut.Error) THEN
					bMPGZAAxisGearOut:=FALSE;
					nMPG_A_State := nMPG_A_State+1;
				ELSIF bMPGZAAxisGearOut AND fbMPGZAAxisGearOut.Error THEN
					bMPGZAAxisGearOut:=FALSE;
					nMPGA_ErrorID := fbMPGZAAxisGearOut.ErrorID;
					nMPG_A_State:=4;
				ELSE
					bMPGZAAxisGearOut:=TRUE;
				END_IF

			4:	(* Request Axis Stop *)
				IF bZAStop AND fbZAAxisStop.Done	AND NOT(fbZAAxisStop.Error) THEN
					bZAStop:=FALSE;
					nMPG_A_State:=nMPG_A_State+1;
				ELSIF bZAStop AND fbZAAxisStop.Error THEN
					bZAStop:=FALSE;
					nMPG_A_State:=5;
				ELSE
					bZAStop:=TRUE;
				END_IF

			5:	(* Fault/Clean Up State *)
				bZAStop:=FALSE;
				bMPGZAAxisGearIn:=FALSE;
				bMPGZAAxisGearOut:=FALSE;
				IF NOT(bZAAxisSelected) THEN
					nMPG_A_State:=0;
					MPGMode := 0;
				END_IF
			END_CASE	(* ZA *)

		4: (* WA Axis Selected *)
			CASE nMPG_A_State OF
			0:	(* INIT *)
				IF NOT bWAAxisSelected THEN
					MPGMode := 0;
				ELSE
					nMPG_A_State := nMPG_A_State + 1;
				END_IF

			1:	(* Request Gear In *)
				IF bMPGWAAxisGearIn AND fbMPGWAAxisGearIn.InGear THEN
					nMPG_A_State:=nMPG_A_State+1;
				ELSIF bMPGWAAxisGearIn AND fbMPGWAAxisGearIn.Error THEN
					bMPGWAAxisGearIn := FALSE;
					nMPGA_ErrorID := fbMPGWAAxisGearIn.ErrorID;
					nMPG_A_State := 5;
				ELSE
					bMPGWAAxisGearIn:=TRUE;
				END_IF

			2:	(* Wait for Axis Selector Change or end if a Fault Occurs *)
				IF NOT(bWAAxisSelected) OR bMachineFault THEN
					nMPG_A_State:=nMPG_A_State+1;
				END_IF

			3:	(* Request Gear Out *)
				IF bMPGWAAxisGearOut AND fbMPGWAAxisGearOut.Done AND NOT(fbMPGWAAxisGearOut.Error) THEN
					bMPGWAAxisGearOut:=FALSE;
					nMPG_A_State := nMPG_A_State+1;
				ELSIF bMPGWAAxisGearOut AND fbMPGWAAxisGearOut.Error THEN
					bMPGWAAxisGearOut:=FALSE;
					nMPGA_ErrorID := fbMPGWAAxisGearOut.ErrorID;
					nMPG_A_State:=4;
				ELSE
					bMPGWAAxisGearIn:=FALSE;
					bMPGWAAxisGearOut:=TRUE;
				END_IF

			4:	(* Request Axis Stop *)
				IF bWAStop AND fbWAAxisStop.Done AND NOT(fbWAAxisStop.Error) THEN
					bWAStop:=FALSE;
					nMPG_A_State:=nMPG_A_State+1;
				ELSIF bWAStop AND fbWAAxisStop.Error THEN
					bWAStop:=FALSE;
					nMPG_A_State:=5;
				ELSE
					bWAStop:=TRUE;
				END_IF

			5:	(* Fault/Clean Up State *)
				bWAStop:=FALSE;
				bMPGWAAxisGearIn:=FALSE;
				bMPGWAAxisGearOut:=FALSE;
				IF NOT(bWAAxisSelected) THEN
					nMPG_A_State:=0;
					MPGMode := 0;
				END_IF
			END_CASE	(* WA *)

		5: (* XB Axis Selected *)
			CASE nMPG_B_State OF
			0:	(* INIT *)
				IF NOT bXBAxisSelected THEN
					MPGMode := 0;
				ELSE
					nMPG_B_State := nMPG_B_State + 1;
				END_IF

			1:	(* Request Gear In *)
				IF bMPGXBAxisGearIn AND fbMPGXBAxisGearIn.InGear THEN
					nMPG_B_State:=nMPG_B_State+1;
				ELSIF bMPGXBAxisGearIn AND fbMPGXBAxisGearIn.Error THEN
					bMPGXBAxisGearIn := FALSE;
					nMPGB_ErrorID := fbMPGXBAxisGearIn.ErrorID;
					nMPG_B_State := 5;
				ELSE
					bMPGXBAxisGearIn:=TRUE;
				END_IF

			2:	(* Wait for Axis Selector Change or end if a Fault Occurs *)
				IF NOT(bXBAxisSelected) OR bMachineFault THEN
					nMPG_B_State:=nMPG_B_State+1;
				END_IF

			3:	(* Request Gear Out *)
				IF bMPGXBAxisGearOut AND fbMPGXBAxisGearOut.Done AND NOT(fbMPGXBAxisGearOut.Error) THEN
					bMPGXBAxisGearOut:=FALSE;
					nMPG_B_State := nMPG_B_State+1;
				ELSIF bMPGXBAxisGearOut AND fbMPGXBAxisGearOut.Error THEN
					bMPGXBAxisGearOut:=FALSE;
					nMPGB_ErrorID := fbMPGXBAxisGearOut.ErrorID;
					nMPG_B_State:=4;
				ELSE
					bMPGXBAxisGearIn:=FALSE;
					bMPGXBAxisGearOut:=TRUE;
				END_IF

			4:	(* Request Axis Stop *)
				IF bUStop AND fbUAxisStop.Done AND NOT(fbUAxisStop.Error) THEN
					bUStop:=FALSE;
					nMPG_B_State:=nMPG_B_State+1;
				ELSIF bUStop AND fbUAxisStop.Error THEN
					bUStop:=FALSE;
					nMPG_B_State:=5;
				ELSE
					bUStop:=TRUE;
				END_IF

			5:	(* Fault/Clean Up State *)
				bUStop:=FALSE;
				bMPGXBAxisGearIn:=FALSE;
				bMPGXBAxisGearOut:=FALSE;
				IF NOT(bXBAxisSelected) THEN
					nMPG_B_State:=0;
					MPGMode := 0;
				END_IF
			END_CASE	(* XB *)

		7: (* ZB Axis Selected *)
			CASE nMPG_B_State OF
			0:	(* INIT *)
				IF NOT bZBAxisSelected THEN
					MPGMode := 0;
				ELSE
					nMPG_B_State := nMPG_B_State + 1;
				END_IF

			1:	(* Request Gear In *)
				IF bMPGZBAxisGearIn AND fbMPGZBAxisGearIn.InGear THEN
					nMPG_B_State:=nMPG_B_State+1;
				ELSIF bMPGZBAxisGearIn AND fbMPGZBAxisGearIn.Error THEN
					bMPGZBAxisGearIn := FALSE;
					nMPGB_ErrorID := fbMPGZBAxisGearIn.ErrorID;
					nMPG_B_State := 5;
				ELSE
					bMPGZBAxisGearIn:=TRUE;
				END_IF

			2:	(* Wait for Axis Selector Change or end if a Fault Occurs *)
				IF NOT(bZBAxisSelected) OR bMachineFault THEN
					bMPGZBAxisGearIn:=FALSE;
					nMPG_B_State:=nMPG_B_State+1;
				END_IF

			3:	(* Request Gear Out *)
				IF bMPGZBAxisGearOut AND fbMPGZBAxisGearOut.Done AND NOT(fbMPGZBAxisGearOut.Error) THEN
					bMPGZBAxisGearOut:=FALSE;
					nMPG_B_State := nMPG_B_State+1;
				ELSIF bMPGZBAxisGearOut AND fbMPGZBAxisGearOut.Error THEN
					bMPGZBAxisGearOut:=FALSE;
					nMPGB_ErrorID := fbMPGZBAxisGearOut.ErrorID;
					nMPG_B_State:=4;
				ELSE
					bMPGZBAxisGearOut:=TRUE;
				END_IF

			4:	(* Request Axis Stop *)
				IF bZBStop AND fbZBAxisStop.Done	AND NOT(fbZBAxisStop.Error) THEN
					bZBStop:=FALSE;
					nMPG_B_State:=nMPG_B_State+1;
				ELSIF bZBStop AND fbZBAxisStop.Error THEN
					bZBStop:=FALSE;
					nMPG_B_State:=5;
				ELSE
					bZBStop:=TRUE;
				END_IF

			5:	(* Fault/Clean Up State *)
				bZBStop:=FALSE;
				bMPGZBAxisGearIn:=FALSE;
				bMPGZBAxisGearOut:=FALSE;
				IF NOT(bZBAxisSelected) THEN
					nMPG_B_State:=0;
					MPGMode := 0;
				END_IF
			END_CASE	(* ZB *)

		8: (* WB Axis Selected *)
			CASE nMPG_B_State OF
			0:	(* INIT *)
				IF NOT bWBAxisSelected THEN
					MPGMode := 0;
				ELSE
					nMPG_B_State := nMPG_B_State + 1;
				END_IF

			1:	(* Request Gear In *)
				IF bMPGWBAxisGearIn AND fbMPGWBAxisGearIn.InGear THEN
					nMPG_B_State:=nMPG_B_State+1;
				ELSIF bMPGWBAxisGearIn AND fbMPGWBAxisGearIn.Error THEN
					bMPGWBAxisGearIn := FALSE;
					nMPGB_ErrorID := fbMPGWBAxisGearIn.ErrorID;
					nMPG_B_State := 5;
				ELSE
					bMPGWBAxisGearIn:=TRUE;
				END_IF

			2:	(* Wait for Axis Selector Change or end if a Fault Occurs *)
				IF NOT(bWBAxisSelected) OR bMachineFault THEN
					nMPG_B_State:=nMPG_B_State+1;
				END_IF

			3:	(* Request Gear Out *)
				IF bMPGWBAxisGearOut AND fbMPGWBAxisGearOut.Done AND NOT(fbMPGWBAxisGearOut.Error) THEN
					bMPGWBAxisGearOut:=FALSE;
					nMPG_B_State := nMPG_B_State+1;
				ELSIF bMPGWBAxisGearOut AND fbMPGWBAxisGearOut.Error THEN
					bMPGWBAxisGearOut:=FALSE;
					nMPGB_ErrorID := fbMPGWBAxisGearOut.ErrorID;
					nMPG_B_State:=4;
				ELSE
					bMPGWBAxisGearIn:=FALSE;
					bMPGWBAxisGearOut:=TRUE;
				END_IF

			4:	(* Request Axis Stop *)
				IF bWBStop AND fbWBAxisStop.Done AND NOT(fbWBAxisStop.Error) THEN
					bWBStop:=FALSE;
					nMPG_B_State:=nMPG_B_State+1;
				ELSIF bWBStop AND fbWBAxisStop.Error THEN
					bWBStop:=FALSE;
					nMPG_B_State:=5;
				ELSE
					bWBStop:=TRUE;
				END_IF

			5:	(* Fault/Clean Up State *)
				bWBStop:=FALSE;
				bMPGWBAxisGearIn:=FALSE;
				bMPGWBAxisGearOut:=FALSE;
				IF NOT(bWBAxisSelected) THEN
					nMPG_B_State:=0;
					MPGMode := 0;
				END_IF
			END_CASE	(* WB *)

	END_CASE	(* Check for MPG Selection *)

ELSE (* Auto Mode or MCC_S is out *)
	bMPGUAAxisGearIn := FALSE;
	bMPGZAAxisGearIn := FALSE;
	bMPGWAAxisGearIn := FALSE;
	bMPGXBAxisGearIn:=FALSE;
	bMPGZBAxisGearIn:=FALSE;
	bMPGWBAxisGearIn:=FALSE;

	bMPGUAAxisGearOut := TRUE;
	bMPGZAAxisGearOut := TRUE;
	bMPGWAAxisGearOut := TRUE;
	bMPGXBAxisGearOut := TRUE;
	bMPGZBAxisGearOut := TRUE;
	bMPGWBAxisGearOut := TRUE;

END_IF

(* Set the Side A MPG Rate by the Selector Switch Input *)
IF bARate1X THEN
	MPG_A_Rate := 1;
ELSIF bARate10X THEN
	MPG_A_Rate := 10;
ELSIF bARate100X THEN
	MPG_A_Rate := 100;
END_IF

(* Set the Side B MPG Rate by the Selector Switch Input *)
IF bBRate1X THEN
	MPG_B_Rate := 1;
ELSIF bBRate10X THEN
	MPG_B_Rate := 10;
ELSIF bBRate100X THEN
	MPG_B_Rate := 100;
END_IF

(*		SIDE A 	 MPG		*)
fbMPGUAOn(CLK:= bXAAxisSelected AND fbAAxisSelectDelay.Q);
fbMPGYAOn(CLK:= bYAAxisSelected AND fbAAxisSelectDelay.Q);
fbMPGZAOn(CLK:= bZAAxisSelected AND fbAAxisSelectDelay.Q);
fbMPGWAOn(CLK:= bWAAxisSelected AND fbAAxisSelectDelay.Q);
fbAAxisSelectDelay(IN:= (bWAAxisSelected XOR bXAAxisSelected XOR bYAAxisSelected XOR bZAAxisSelected)
, PT:=t#500ms);

fbMPGAAxisEnable(
	Enable:=bMPGAAxisEnable ,
	Enable_Positive:= bMPGAAxisEnable ,
	Enable_Negative:= bMPGAAxisEnable ,
	Override:=100 ,
	BufferMode:=MC_Aborting ,
	Axis := stAxisMPG_A );

fGearRatioA := MPG_A_Rate/100.0;

fbMPGUAAxisGearIn(
	Enable:= bMPGUAAxisGearIn ,
	GearRatio:= -fGearRatioA ,
	Acceleration:=0 ,
	Deceleration:=0 ,
	Jerk:=0 ,
	Master := stAxisMPG_A ,
	Slave := stUAxis
);

fbMPGUAAxisGearOut(
	Execute := bMPGUAAxisGearOut ,
	Slave := stUAxis
);

fbMPGWAAxisGearIn(
	Enable:= bMPGWAAxisGearIn ,
	GearRatio:= -fGearRatioA ,
	Acceleration:=0 ,
	Deceleration:=0 ,
	Jerk:=0 ,
	Master := stAxisMPG_A ,
	Slave := stWAAxis
);

fbMPGWAAxisGearOut(
	Execute := bMPGWAAxisGearOut ,
	Slave := stWAAxis
);

fbMPGZAAxisGearIn(
	Enable:= bMPGZAAxisGearIn ,
	GearRatio:= -fGearRatioA ,
	Acceleration:=0 ,
	Deceleration:=0 ,
	Jerk:=0 ,
	Master := stAxisMPG_A ,
	Slave := stZAAxis
);

fbMPGZAAxisGearOut(
	Execute:= bMPGZAAxisGearOut ,
	Slave:=stZAAxis
);

(*		SIDE B		 MPG		*)
fbMPGXBOn(CLK:= bXBAxisSelected AND fbBAxisSelectDelay.Q);
fbMPGYBOn(CLK:= bYBAxisSelected AND fbBAxisSelectDelay.Q);
fbMPGZBOn(CLK:= bZBAxisSelected AND fbBAxisSelectDelay.Q);
fbMPGWBOn(CLK:= bWBAxisSelected AND fbBAxisSelectDelay.Q);
fbBAxisSelectDelay(IN:= (bWBAxisSelected XOR bXBAxisSelected XOR bYBAxisSelected XOR bZBAxisSelected)
, PT:=t#500ms);

fbMPGBAxisEnable(
	Enable:=bMPGBAxisEnable ,
	Enable_Positive:= bMPGBAxisEnable ,
	Enable_Negative:= bMPGBAxisEnable ,
	Override:=100 ,
	BufferMode:=MC_Aborting ,
	Axis := stAxisMPG_B );

fGearRatioB := MPG_B_Rate/100.0;

fbMPGWBAxisGearIn(
	Enable:= bMPGWBAxisGearIn ,
	GearRatio:= -fGearRatioB ,
	Acceleration:=0 ,
	Deceleration:=0 ,
	Jerk:=0 ,
	Master := stAxisMPG_B ,
	Slave := stWBAxis
);

fbMPGWBAxisGearOut(
	Execute := bMPGWBAxisGearOut ,
	Slave := stWBAxis
);

fbMPGXBAxisGearIn(
	Enable:= bMPGXBAxisGearIn ,
	GearRatio:= -fGearRatioB ,
	Acceleration:=0 ,
	Deceleration:=0 ,
	Jerk:=0 ,
	Master := stAxisMPG_B ,
	Slave := stUAxis
);

fbMPGXBAxisGearOut(
	Execute := bMPGXBAxisGearOut ,
	Slave := stUAxis
);

fbMPGZBAxisGearIn(
	Enable:= bMPGZBAxisGearIn ,
	GearRatio:= -fGearRatioB ,
	Acceleration:=0 ,
	Deceleration:=0 ,
	Jerk:=0 ,
	Master := stAxisMPG_B ,
	Slave := stZBAxis
);

fbMPGZBAxisGearOut(
	Execute:= bMPGZBAxisGearOut ,
	Slave:=stZBAxis
);


(* Reset the MPG Axis *)
IF fbMPGAAxisMCReset.Done OR fbMPGAAxisMCReset.Error THEN
	bMPGA_MCResetRequest:=FALSE;
END_IF
fbMPGAAxisMCReset(
	Execute:=bMPGA_MCResetRequest,
	Axis:=stAxisMPG_A );

IF fbMPGBAxisMCReset.Done OR fbMPGBAxisMCReset.Error THEN
	bMPGB_MCResetRequest:=FALSE;
END_IF
fbMPGBAxisMCReset(
	Execute:=bMPGB_MCResetRequest,
	Axis:=stAxisMPG_B );

fbMPGWatchdog(IN:=bMPGWatchdog, PT:= t#150ms);
fbMPGBWatchdog(IN:=bMPGBWatchdog, PT:= t#150ms);
END_PROGRAM

(* POU Programs/Build_Send_Network_Data, ST *)
PROGRAM Build_Send_Network_Data
(* The program translates the values recieved in the Structure ST_Panel_Receive arrays and places it into the values to be displayed on the screens *)
VAR
	fbHistoryElementTimer: TON;		(* timer to trigger a different Element of the Fault History to pass to the Panels *)
	nHistoryElement : INT := 1;			(* Fault History Element # to pass to the Panels *)
END_VAR
(* Miscellaneous Variables to Send *)

	(* Boolian variaables to Send *)
	stCXPublish1.arrBOOL[1] := bMachineFault ;
	stCXPublish1.arrBOOL[2] := bMachineWarning;
	stCXPublish1.arrBOOL[3] := bCoolantTempWarning;
	stCXPublish1.arrBOOL[4] := bCoolantTempFault;
	stCXPublish1.arrBOOL[5] := bMachineMode;
	stCXPublish1.arrBOOL[6] := bInCycle;

	(* Send the Fault Message Array *)
	stCXPublish1.arrSTRING50[1] := arrFaultMessage[1];
	stCXPublish1.arrSTRING50[2] := arrFaultMessage[2];
	stCXPublish1.arrSTRING50[3] := arrFaultMessage[3];
	stCXPublish1.arrSTRING50[4] := arrFaultMessage[4];
	stCXPublish1.arrSTRING50[5] := arrFaultMessage[5];
	stCXPublish1.arrSTRING50[6] := arrFaultMessage[6];
	stCXPublish1.arrSTRING50[7] := arrFaultMessage[7];
	stCXPublish1.arrSTRING50[8] := arrFaultMessage[8];
	stCXPublish1.arrSTRING50[9] := arrFaultMessage[9];
	stCXPublish1.arrSTRING50[10] := arrFaultMessage[10];

	(* Send the Fault History Array to the panels.  One Variable at a time *)
	fbHistoryElementTimer(IN:=TRUE, PT:=t#300ms);
	(* Every 1/2 second we incriment the Element to be sent *)
	IF fbHistoryElementTimer.Q THEN
		fbHistoryElementTimer(IN:=FALSE);
		nHistoryElement:=nHistoryElement+1;
		(* If we are greater than 80 then reset to 1 *)
		IF nHistoryElement > 80 THEN
			nHistoryElement:=1;
		END_IF
	END_IF
	stCXPublish1.arrUDINTIGER[43] := nHistoryElement;
	stCXPublish1.arrSTRING50[11] := arrFaultHistory[nHistoryElement];

	stCXPublish1.arrUDINTIGER[27] := nAutoCycleStep;
	stCXPublish1.arrUDINTIGER[28] := nEtherCATMasterState;
	stCXPublish1.arrUDINTIGER[42] := nAutoModeState;

	(* Security *)
	arrMachineInfo[10] := sUsername;
	arrMachineInfo[11] := sPassword;
	arrMachineInfo[12] := sSavePassword;
	stCXPublish1.arrUDINTIGER[40] := CurrentUserLevel;
	stCXPublish1.arrBOOL[7] := bWrongPassword;
	stCXPublish1.arrBOOL[69] := bWrongSavePassword;

(***** SECRET Screen Variables to Send *)
	(* LREAL  Variables to Send *)
	stCXPublish1.arrUDINTIGER[29] := nUAxisThrustMax;
	stCXPublish1.arrUDINTIGER[36] := nTailstockClampingTorqueLimit;
	stCXPublish1.arrLREAL[35] := fWAAxisHomeOffset;
	stCXPublish1.arrLREAL[36] := fWBAxisHomeOffset;
	stCXPublish1.arrLREAL[37] := fWAxisMoveOffBushing;
	stCXPublish1.arrLREAL[38] := fTailstockVelocity;
	arrMachineInfo[7] := sLoadSideSet;
	stCXPublish1.arrBOOL[8] := bSideAEnabled;
	stCXPublish1.arrBOOL[9] := bSideBEnabled;

(***** MAIN SCREEN Variables to Send *)
	(* Main Screen *)
	arrMachineInfo[1] := sSerialNumber;
	arrMachineInfo[2] := sKaysJobNumber;
	arrMachineInfo[3] := sModelNumber;
	arrMachineInfo[4] := sCustomerName;
	arrMachineInfo[5] := sProductionDate;
	(* Get Current CX Program Program *)
	arrMachineInfo[6] := CONCAT(UDINT_TO_STRING(F_GetVersionDehoff(1)), '.   ');
	arrMachineInfo[6] := CONCAT(arrMachineInfo[6], UDINT_TO_STRING(F_GetVersionDehoff(2)) );

	(* UDINT Variables to Send *)
	stCXPublish1.arrUDINTIGER[20] := nMotorNominalRPM;
	stCXPublish1.arrUDINTIGER[21] := nMachineNumber;

	stCXPublish1.arrUDINTIGER[22] := nFaultArrayIndex;
	stCXPublish1.arrUDINTIGER[23] := nWarningArrayIndex;

	stCXPublish1.arrBOOL[66] := bUserNameHandshake;
	stCXPublish1.arrBOOL[67] := bPasswordHandshake;
	stCXPublish1.arrBOOL[68] := bSavePasswordHandshake;

(*********		PART PROGRAM Variables	  ***********)
(* These variaables are only published when a panel is on the Part Program Screen *)
	stPartProgramSend.arrLREAL[1] := fStartFeed ;
	stPartProgramSend.arrLREAL[2] := fFinishFeed;
	stPartProgramSend.arrLREAL[3] := fStartDepth;
	stPartProgramSend.arrLREAL[4] := fFinishDepth;
	stPartProgramSend.arrLREAL[5] := fDwellTime;
	stPartProgramSend.arrLREAL[6] := fRetractRate;
	stPartProgramSend.arrLREAL[7] := fDrillTipOffset;
	stPartProgramSend.arrLREAL[8] := fRPMRequest;
	stPartProgramSend.arrLREAL[9] := fToolDiameter;
	stPartProgramSend.arrLREAL[10] := fCoolantPressure;
	stPartProgramSend.arrLREAL[11] := fCoolantFlowMax;
	stPartProgramSend.arrLREAL[12] := fCoolantFlowMin;

	stPartProgramSend.arrBOOL[1] := bSpindleRetractMode;
	stPartProgramSend.arrBOOL[2] := bStartFeedChanged;
	stPartProgramSend.arrBOOL[3] := bFinishFeedChanged;
	stPartProgramSend.arrBOOL[4] := bStartDepthChanged;
	stPartProgramSend.arrBOOL[5] := bFinishDepthChanged;
	stPartProgramSend.arrBOOL[6] := bDwellTimeChanged;
	stPartProgramSend.arrBOOL[7] := bRetractRateChanged;
	stPartProgramSend.arrBOOL[8] := bDrillTipOffsetChanged;
	stPartProgramSend.arrBOOL[9] := bRPMRequestChanged;
	stPartProgramSend.arrBOOL[10] := bSpindleRetractChanged;
	stPartProgramSend.arrBOOL[11] := bToolDiameterChanged;
	stPartProgramSend.arrBOOL[12] := bSpindleLoadMaxChanged;
	stPartProgramSend.arrBOOL[13] := bServoThrustMaxChanged;
	stPartProgramSend.arrBOOL[14] := bCoolantFlowMaxChanged;
	stPartProgramSend.arrBOOL[15] := bCoolantFlowMinChanged;
	stPartProgramSend.arrBOOL[16] := bMaxCyclesChanged;

	stPartProgramSend.arrSTRING[1] := sLastLoadedPartProgramName;
	stPartProgramSend.arrSTRING[2] := sFileOpError;
	stPartProgramSend.arrSTRING[3] := sPartProgramName;
	stPartProgramSend.arrSTRING[4] := sCurrentPartProgram;

	stCXPublish1.arrUDINTIGER[24] := nMaxCycles;				(* On Auto Also *)
	stCXPublish1.arrUDINTIGER[25] := nSpindleLoadMax;			(* On Auto Also *)
	stCXPublish1.arrUDINTIGER[26] := nServoThrustMax;			(* On Auto Also *)

(*********		AUTO SCREEN DISPLAY VARIABLES **********)
	(* UDINT Variables to Send *)
	stCXPublish1.arrUDINTIGER[1] := nCycleTimeMinutes;
	stCXPublish1.arrUDINTIGER[2] := nCycleTimeSeconds;
	stCXPublish1.arrUDINTIGER[3] := nCyclesComplete;
	stCXPublish1.arrUDINTIGER[4] := nPartsCompleteTotal;
	stCXPublish1.arrUDINTIGER[37] := nPartsCompleteA1;
	stCXPublish1.arrUDINTIGER[38] := nPartsCompleteA2;
	stCXPublish1.arrUDINTIGER[39] := nPartsCompleteA3;
	stCXPublish1.arrUDINTIGER[32] := nPartsCompleteB1;
	stCXPublish1.arrUDINTIGER[35] := nPartsCompleteB2;
	stCXPublish1.arrUDINTIGER[41] := nPartsCompleteB3;

	stCXPublish1.arrUDINTIGER[5] := nSpindleRPM1A;
	stCXPublish1.arrUDINTIGER[6] := nSpindleRPM2A;
	stCXPublish1.arrUDINTIGER[7] := nSpindleRPM3A;
	stCXPublish1.arrUDINTIGER[8] := nSpindleRPM1B;
	stCXPublish1.arrUDINTIGER[9] := nSpindleRPM2B;
	stCXPublish1.arrUDINTIGER[10] := nSpindleRPM3B;
	nSpindleLoad1ADisplay:=LREAL_TO_UDINT(
		stVFD_A1DriveInfo.fMotorCurrent / stVFD_A1DriveInfo.fMotorNominalCurrent * 100);
	stCXPublish1.arrUDINTIGER[11] := nSpindleLoad1ADisplay;
	nSpindleLoad2ADisplay:=LREAL_TO_UDINT(
		stVFD_A2DriveInfo.fMotorCurrent / stVFD_A2DriveInfo.fMotorNominalCurrent * 100);
	stCXPublish1.arrUDINTIGER[12] := nSpindleLoad2ADisplay;
	nSpindleLoad3ADisplay:=LREAL_TO_UDINT(
		stVFD_A3DriveInfo.fMotorCurrent / stVFD_A3DriveInfo.fMotorNominalCurrent * 100);
	stCXPublish1.arrUDINTIGER[13] := nSpindleLoad3ADisplay;
	nSpindleLoad1BDisplay:=LREAL_TO_UDINT(
		stVFD_B1DriveInfo.fMotorCurrent / stVFD_B1DriveInfo.fMotorNominalCurrent * 100);
	stCXPublish1.arrUDINTIGER[14] := nSpindleLoad1BDisplay;
	nSpindleLoad2BDisplay:=LREAL_TO_UDINT(
		stVFD_B2DriveInfo.fMotorCurrent / stVFD_B2DriveInfo.fMotorNominalCurrent * 100);
	stCXPublish1.arrUDINTIGER[15] := nSpindleLoad2BDisplay;
	nSpindleLoad3BDisplay:=LREAL_TO_UDINT(
		stVFD_B3DriveInfo.fMotorCurrent / stVFD_B3DriveInfo.fMotorNominalCurrent * 100);
	stCXPublish1.arrUDINTIGER[16] := nSpindleLoad3BDisplay;

	(*	Servo Thrust Display Conversion *)
	IF bAServoEnable THEN
		nServoAThrustDisplay:=ABS(LREAL_TO_DINT(nServoZAThrust/10.0));
	ELSE
		nServoAThrustDisplay:=0;
	END_IF
	stCXPublish1.arrUDINTIGER[17] := nServoAThrustDisplay;

	IF bBServoEnable THEN
		nServoBThrustDisplay:=ABS(LREAL_TO_DINT(nServoZBThrust/10.0));
	ELSE
		nServoBThrustDisplay:=0;
	END_IF
	stCXPublish1.arrUDINTIGER[18] := nServoBThrustDisplay;

	(* LREAL  Variables to Send *)
	stCXPublish1.arrLREAL[1] := fCoolantTempDisplay;

	fCoolantFlow1ADisplay:=(nCoolantFlowA1/32767.0*(fFlowMonitorMax));
	stCXPublish1.arrLREAL[2] := fCoolantFlow1ADisplay;
	fCoolantFlow1AGraph:=nCoolantFlowA1/32767.0*100;
	stCXPublish1.arrLREAL[3] := fCoolantFlow1AGraph;
	fCoolantFlow2ADisplay:=(nCoolantFlowA2/32767.0*(fFlowMonitorMax));
	stCXPublish1.arrLREAL[4] := fCoolantFlow2ADisplay;
	fCoolantFlow2AGraph:=nCoolantFlowA2/32767.0*100;
	stCXPublish1.arrLREAL[5] := fCoolantFlow2AGraph;
	fCoolantFlow3ADisplay:=(nCoolantFlowA3/32767.0*(fFlowMonitorMax));
	stCXPublish1.arrLREAL[6] := fCoolantFlow3ADisplay;
	fCoolantFlow3AGraph:=nCoolantFlowA3/32767.0*100;
	stCXPublish1.arrLREAL[7] := fCoolantFlow3AGraph;

	fCoolantFlow1BDisplay:=(nCoolantFlowB1/32767.0*(fFlowMonitorMax));
	stCXPublish1.arrLREAL[8] 	:= fCoolantFlow1BDisplay;
	fCoolantFlow1BGraph:=nCoolantFlowB1/32767.0*100;
	stCXPublish1.arrLREAL[9] 	:= fCoolantFlow1BGraph;
	fCoolantFlow2BDisplay:=(nCoolantFlowB2/32767.0*(fFlowMonitorMax));
	stCXPublish1.arrLREAL[10] 	:= fCoolantFlow2BDisplay;
	fCoolantFlow2BGraph:=nCoolantFlowB2/32767.0*100;
	stCXPublish1.arrLREAL[11] 	:= fCoolantFlow2BGraph;
	fCoolantFlow3BDisplay:=(nCoolantFlowB3/32767.0*(fFlowMonitorMax));
	stCXPublish1.arrLREAL[12] 	:= fCoolantFlow3BDisplay;
	fCoolantFlow3BGraph:=nCoolantFlowB3/32767.0*100;
	stCXPublish1.arrLREAL[13] 	:= fCoolantFlow3BGraph;

	fZAAxisVelosity 			:= stZAAxis.NcToPlc.SetVelo*60;
	stCXPublish1.arrLREAL[14] 	:= fZAAxisVelosity;
	fZBAxisVelosity 			:= stZBAxis.NcToPlc.SetVelo*60;
	stCXPublish1.arrLREAL[15] 	:= fZBAxisVelosity;

	stCXPublish1.arrLREAL[16] := stZAAxis.NcToPlc.ActPos;
	stCXPublish1.arrLREAL[17] := stZBAxis.NcToPlc.ActPos;
	stCXPublish1.arrLREAL[18] := stWAAxis.NcToPlc.ActPos;
	stCXPublish1.arrLREAL[19] := stWBAxis.NcToPlc.ActPos;

	fFlowMonitorMax := 60;
	stCXPublish1.arrLREAL[20] 	:= fFlowMonitorMax;
	fCoolantFlowMinGraph 		:= fCoolantFlowMin/fFlowMonitorMax*100.0;
	stCXPublish1.arrLREAL[21] 	:= fCoolantFlowMinGraph;
	fCoolantFlowMaxGraph 	:= 100-(fCoolantFlowMax/fFlowMonitorMax*100.0);
	stCXPublish1.arrLREAL[22] 	:= fCoolantFlowMaxGraph;

	stCXPublish1.arrBOOL[63] 	:= bCellRunOutRequest;
	stCXPublish1.arrBOOL[64]	:= bDisplayUnloadConf;
	stCXPublish1.arrBOOL[65]	:= bDispPressCycleStart;


(*********		TRANSFER SCREEN DISPLAY VARIABLES **********)
	stCXPublish1.arrLREAL[25] := stUAxis.NcToPlc.ActPos;
	IF (sLoadSideSet = 'A') THEN
		stCXPublish1.arrLREAL[26] := fUAxisLoadSidePosition;
		stCXPublish1.arrLREAL[27]:= fUAxisUnloadSidePosition;
	ELSIF  (sLoadSideSet = 'B') THEN
		stCXPublish1.arrLREAL[27] := fUAxisLoadSidePosition;
		stCXPublish1.arrLREAL[26]:= fUAxisUnloadSidePosition;
	END_IF
	stCXPublish1.arrLREAL[28]:= fUAxisVelocity;

	stCXPublish1.arrBOOL[10] := stUAxis.NcToPlc.StateDWord.1;
	stCXPublish1.arrBOOL[11] := bProx516;
	stCXPublish1.arrBOOL[12] := bProx517;
	stCXPublish1.arrBOOL[13] := bTransferUp;
	stCXPublish1.arrBOOL[14] := bTransferDown;
	stCXPublish1.arrBOOL[15] := bProx410;
	stCXPublish1.arrBOOL[16] := bProx411;
	stCXPublish1.arrBOOL[17] := bProx412;
	stCXPublish1.arrBOOL[18] := bProx413;
	stCXPublish1.arrBOOL[19] := bProx414;
	stCXPublish1.arrBOOL[20] := bProx415;
	stCXPublish1.arrBOOL[21] := bProx510;
	stCXPublish1.arrBOOL[22] := bProx511;
	stCXPublish1.arrBOOL[23] := bProx512;
	stCXPublish1.arrBOOL[24] := bProx513;
	stCXPublish1.arrBOOL[25] := bProx514;
	stCXPublish1.arrBOOL[26] := bProx515;
	stCXPublish1.arrBOOL[27] := bTransferAtLoadIndicator;

(*********		FIXTURE SCREEN DISPLAY VARIABLES **********)
	stCXPublish1.arrLREAL[30] := fWAxisTransferPosition;
	stCXPublish1.arrLREAL[31] := fWAxisDrillPosition;

	(* A Side *)
	stCXPublish1.arrUDINTIGER[30] := nWAAxisThrust;
	stCXPublish1.arrUDINTIGER[31] := nWAAxisThrustMax;

	stCXPublish1.arrBOOL[30] := stWAAxis.NcToPlc.StateDWord.1;
	stCXPublish1.arrBOOL[31] := bPS616;
	stCXPublish1.arrBOOL[32] := bPS617;
	stCXPublish1.arrBOOL[33] := bProx610;
	stCXPublish1.arrBOOL[34] := bProx611;
	stCXPublish1.arrBOOL[35] := bProx612;
	stCXPublish1.arrBOOL[36] := bProx613;
	stCXPublish1.arrBOOL[37] := bProx614;
	stCXPublish1.arrBOOL[38] := bProx615;
	stCXPublish1.arrBOOL[39] := bAEjectorOvertravelError;

	(* B Side *)
	stCXPublish1.arrUDINTIGER[33] := nWBAxisThrust;
	stCXPublish1.arrUDINTIGER[34] := nWBAxisThrustMax;

	stCXPublish1.arrBOOL[40] := stWBAxis.NcToPlc.StateDWord.1;
	stCXPublish1.arrBOOL[41] := bPS726;
	stCXPublish1.arrBOOL[42] := bPS727;
	stCXPublish1.arrBOOL[43] := bProx720;
	stCXPublish1.arrBOOL[44] := bProx721;
	stCXPublish1.arrBOOL[45] := bProx722;
	stCXPublish1.arrBOOL[46] := bProx723;
	stCXPublish1.arrBOOL[47] := bProx724;
	stCXPublish1.arrBOOL[48] := bProx725;
	stCXPublish1.arrBOOL[49] := bBEjectorOvertravelError;

(**********		MANUAL SCREEN Display Variables	*******)
	stCXPublish1.arrBOOL[50] :=stZAAxis.NcToPlc.StateDWord.1;
	stCXPublish1.arrBOOL[51] :=stZBAxis.NcToPlc.StateDWord.1;
	stCXPublish1.arrBOOL[52] := bHydraulicSystemPressure;
	stCXPublish1.arrBOOL[53] := bHighPressureMotorRunning;
	stCXPublish1.arrBOOL[54] := bTransferPumpMotorRunning;
	stCXPublish1.arrBOOL[55] := bConveyorFWDReq;
	stCXPublish1.arrBOOL[56] := bACoolantSolenoid;
	stCXPublish1.arrBOOL[57] := bBCoolantSolenoid;
	stCXPublish1.arrBOOL[58] := bMCR;
	stCXPublish1.arrBOOL[59] := bMCC_SConfirm;
	stCXPublish1.arrBOOL[60] := bPneumaticSystemPressure;
	stCXPublish1.arrBOOL[61] := bLubePressure;
	stCXPublish1.arrBOOL[62] := bLubeLevel;

(****** 	FAULT Screen 		******)
	stCXPublish1.arrUDINTIGER[46] := nZAAxisDiagNumber ;
	stCXPublish1.arrUDINTIGER[47] := nWAAxisDiagNumber;
	stCXPublish1.arrUDINTIGER[48] := nZBAxisDiagNumber;
	stCXPublish1.arrUDINTIGER[49] := nWBAxisDiagNumber;
	stCXPublish1.arrUDINTIGER[50] := nUAxisDiagNumber;

(******	Test Speed Screen 	*****)
	stCXPublish1.arrUDINTIGER[19] := nTestSpeedOverRide;

	stCXPublish1.arrBOOL[29] := bTestSpeedOn;
END_PROGRAM

